	X =  100.000  mm,	Y =  199.000  mm,	Z =   15.000 mm,
	W =180.000 deg,	P =   0.000 deg,	R =    90.000 deg
};
P[9151]{
   GP1:
	UF : 1, UT : 1,		CONFIG : 'N U T, 0, 0, 1',
	X =  103.000  mm,	Y =  199.000  mm,	Z =   15.000 mm,
	W =180.000 deg,	P =   0.000 deg,	R =    90.000 deg
};
P[9152]{
   GP1:
	UF : 1, UT : 1,		CONFIG : 'N U T, 0, 0, 1',
	X =  103.000  mm,	Y =  199.000  mm,	Z =   0.600 mm,
	W =180.000 deg,	P =   0.000 deg,	R =    90.000 deg
};
P[9153]{
   GP1:
	UF : 1, UT : 1,		CONFIG : 'N U T, 0, 0, 1',
	X =  103.000  mm,	Y =  199.000  mm,	Z =   15.000 mm,
	W =180.000 deg,	P =   0.000 deg,	R =    90.000 deg
};
P[9154]{
   GP1:
	UF : 1, UT : 1,		CONFIG : 'N U T, 0, 0, 1',
	X =  106.000  mm,	Y =  199.000  mm,	Z =   15.000 mm,
	W =180.000 deg,	P =   0.000 deg,	R =    90.000 deg
};
P[9155]{
   GP1:
	UF : 1, UT : 1,		CONFIG : 'N U T, 0, 0, 1',
	X =  106.000  mm,	Y =  199.000  mm,	Z =   0.600 mm,
	W =180.000 deg,	P =   0.000 deg,	R =    90.000 deg
};
P[9156]{
   GP1:
	UF : 1, UT : 1,		CONFIG : 'N U T, 0, 0, 1',
	X =  106.000  mm,	Y =  199.000  mm,	Z =   15.000 mm,
	W =180.000 deg,	P =   0.000 deg,	R =    90.000 deg
};
P[9157]{
   GP1:
	UF : 1, UT : 1,		CONFIG : 'N U T, 0, 0, 1',
	X =  109.000  mm,	Y =  199.000  mm,	Z =   15.000 mm,
	W =180.000 deg,	P =   0.000 deg,	R =    90.000 deg
};
P[9158]{
   GP1:
	UF : 1, UT : 1,		CONFIG : 'N U T, 0, 0, 1',
	X =  109.000  mm,	Y =  199.000  mm,	Z =   0.600 mm,
	W =180.000 deg,	P =   0.000 deg,	R =    90.000 deg
};
P[9159]{
   GP1:
	UF : 1, UT : 1,		CONFIG : 'N U T, 0, 0, 1',
	X =  109.000  mm,	Y =  199.000  mm,	Z =   15.000 mm,
	W =180.000 deg,	P =   0.000 deg,	R =    90.000 deg
};
P[9160]{
   GP1:
	UF : 1, UT : 1,		CONFIG : 'N U T, 0, 0, 1',
	X =  112.000  mm,	Y =  199.000  mm,	Z =   15.000 mm,
	W =180.000 deg,	P =   0.000 deg,	R =    90.000 deg
};
P[9161]{
   GP1:
	UF : 1, UT : 1,		CONFIG : 'N U T, 0, 0, 1',
	X =  112.000  mm,	Y =  199.000  mm,	Z =   0.600 mm,
	W =180.000 deg,	P =   0.000 deg,	R =    90.000 deg
};
P[9162]{
   GP1:
	UF : 1, UT : 1,		CONFIG : 'N U T, 0, 0, 1',
	X =  112.000  mm,	Y =  199.000  mm,	Z =   15.000 mm,
	W =180.000 deg,	P =   0.000 deg,	R =    90.000 deg
};
P[9163]{
   GP1:
	UF : 1, UT : 1,		CONFIG : 'N U T, 0, 0, 1',
	X =  115.000  mm,	Y =  199.000  mm,	Z =   15.000 mm,
	W =180.000 deg,	P =   0.000 deg,	R =    90.000 deg
};
P[9164]{
   GP1:
	UF : 1, UT : 1,		CONFIG : 'N U T, 0, 0, 1',
	X =  115.000  mm,	Y =  199.000  mm,	Z =   0.600 mm,
	W =180.000 deg,	P =   0.000 deg,	R =    90.000 deg
};
P[9165]{
   GP1:
	UF : 1, UT : 1,		CONFIG : 'N U T, 0, 0, 1',
	X =  115.000  mm,	Y =  199.000  mm,	Z =   15.000 mm,
	W =180.000 deg,	P =   0.000 deg,	R =    90.000 deg
};
P[9166]{
   GP1:
	UF : 1, UT : 1,		CONFIG : 'N U T, 0, 0, 1',
	X =  118.000  mm,	Y =  199.000  mm,	Z =   15.000 mm,
	W =180.000 deg,	P =   0.000 deg,	R =    90.000 deg
};
P[9167]{
   GP1:
	UF : 1, UT : 1,		CONFIG : 'N U T, 0, 0, 1',
	X =  118.000  mm,	Y =  199.000  mm,	Z =   0.600 mm,
	W =180.000 deg,	P =   0.000 deg,	R =    90.000 deg
};
P[9168]{
   GP1:
	UF : 1, UT : 1,		CONFIG : 'N U T, 0, 0, 1',
	X =  118.000  mm,	Y =  199.000  mm,	Z =   15.000 mm,
	W =180.000 deg,	P =   0.000 deg,	R =    90.000 deg
};
P[9169]{
   GP1:
	UF : 1, UT : 1,		CONFIG : 'N U T, 0, 0, 1',
	X =  121.000  mm,	Y =  199.000  mm,	Z =   15.000 mm,
	W =180.000 deg,	P =   0.000 deg,	R =    90.000 deg
};
P[9170]{
   GP1:
	UF : 1, UT : 1,		CONFIG : 'N U T, 0, 0, 1',
	X =  121.000  mm,	Y =  199.000  mm,	Z =   0.600 mm,
	W =180.000 deg,	P =   0.000 deg,	R =    90.000 deg
};
P[9171]{
   GP1:
	UF : 1, UT : 1,		CONFIG : 'N U T, 0, 0, 1',
	X =  121.000  mm,	Y =  199.000  mm,	Z =   15.000 mm,
	W =180.000 deg,	P =   0.000 deg,	R =    90.000 deg
};
P[9172]{
   GP1:
	UF : 1, UT : 1,		CONFIG : 'N U T, 0, 0, 1',
	X =  124.000  mm,	Y =  199.000  mm,	Z =   15.000 mm,
	W =180.000 deg,	P =   0.000 deg,	R =    90.000 deg
};
P[9173]{
   GP1:
	UF : 1, UT : 1,		CONFIG : 'N U T, 0, 0, 1',
	X =  124.000  mm,	Y =  199.000  mm,	Z =   0.600 mm,
	W =180.000 deg,	P =   0.000 deg,	R =    90.000 deg
};
P[9174]{
   GP1:
	UF : 1, UT : 1,		CONFIG : 'N U T, 0, 0, 1',
	X =  124.000  mm,	Y =  199.000  mm,	Z =   15.000 mm,
	W =180.000 deg,	P =   0.000 deg,	R =    90.000 deg
};
P[9175]{
   GP1:
	UF : 1, UT : 1,		CONFIG : 'N U T, 0, 0, 1',
	X =  127.000  mm,	Y =  199.000  mm,	Z =   15.000 mm,
	W =180.000 deg,	P =   0.000 deg,	R =    90.000 deg
};
P[9176]{
   GP1:
	UF : 1, UT : 1,		CONFIG : 'N U T, 0, 0, 1',
	X =  127.000  mm,	Y =  199.000  mm,	Z =   0.600 mm,
	W =180.000 deg,	P =   0.000 deg,	R =    90.000 deg
};
P[9177]{
   GP1:
	UF : 1, UT : 1,		CONFIG : 'N U T, 0, 0, 1',
	X =  127.000  mm,	Y =  199.000  mm,	Z =   15.000 mm,
	W =180.000 deg,	P =   0.000 deg,	R =    90.000 deg
};
P[9178]{
   GP1:
	UF : 1, UT : 1,		CONFIG : 'N U T, 0, 0, 1',
	X =  130.000  mm,	Y =  199.000  mm,	Z =   15.000 mm,
	W =180.000 deg,	P =   0.000 deg,	R =    90.000 deg
};
P[9179]{
   GP1:
	UF : 1, UT : 1,		CONFIG : 'N U T, 0, 0, 1',
	X =  130.000  mm,	Y =  199.000  mm,	Z =   0.600 mm,
	W =180.000 deg,	P =   0.000 deg,	R =    90.000 deg
};
P[9180]{
   GP1:
	UF : 1, UT : 1,		CONFIG : 'N U T, 0, 0, 1',
	X =  130.000  mm,	Y =  199.000  mm,	Z =   15.000 mm,
	W =180.000 deg,	P =   0.000 deg,	R =    90.000 deg
};
P[9181]{
   GP1:
	UF : 1, UT : 1,		CONFIG : 'N U T, 0, 0, 1',
	X =  133.000  mm,	Y =  199.000  mm,	Z =   15.000 mm,
	W =180.000 deg,	P =   0.000 deg,	R =    90.000 deg
};
P[9182]{
   GP1:
	UF : 1, UT : 1,		CONFIG : 'N U T, 0, 0, 1',
	X =  133.000  mm,	Y =  199.000  mm,	Z =   0.600 mm,
	W =180.000 deg,	P =   0.000 deg,	R =    90.000 deg
};
P[9183]{
   GP1:
	UF : 1, UT : 1,		CONFIG : 'N U T, 0, 0, 1',
	X =  133.000  mm,	Y =  199.000  mm,	Z =   15.000 mm,
	W =180.000 deg,	P =   0.000 deg,	R =    90.000 deg
};
P[9184]{
   GP1:
	UF : 1, UT : 1,		CONFIG : 'N U T, 0, 0, 1',
	X =  136.000  mm,	Y =  199.000  mm,	Z =   15.000 mm,
	W =180.000 deg,	P =   0.000 deg,	R =    90.000 deg
};
P[9185]{
   GP1:
	UF : 1, UT : 1,		CONFIG : 'N U T, 0, 0, 1',
	X =  136.000  mm,	Y =  199.000  mm,	Z =   0.600 mm,
	W =180.000 deg,	P =   0.000 deg,	R =    90.000 deg
};
P[9186]{
   GP1:
	UF : 1, UT : 1,		CONFIG : 'N U T, 0, 0, 1',
	X =  136.000  mm,	Y =  199.000  mm,	Z =   15.000 mm,
	W =180.000 deg,	P =   0.000 deg,	R =    90.000 deg
};
P[9187]{
   GP1:
	UF : 1, UT : 1,		CONFIG : 'N U T, 0, 0, 1',
	X =  139.000  mm,	Y =  199.000  mm,	Z =   15.000 mm,
	W =180.000 deg,	P =   0.000 deg,	R =    90.000 deg
};
P[9188]{
   GP1:
	UF : 1, UT : 1,		CONFIG : 'N U T, 0, 0, 1',
	X =  139.000  mm,	Y =  199.000  mm,	Z =   0.600 mm,
	W =180.000 deg,	P =   0.000 deg,	R =    90.000 deg
};
P[9189]{
   GP1:
	UF : 1, UT : 1,		CONFIG : 'N U T, 0, 0, 1',
	X =  139.000  mm,	Y =  199.000  mm,	Z =   15.000 mm,
	W =180.000 deg,	P =   0.000 deg,	R =    90.000 deg
};
P[9190]{
   GP1:
	UF : 1, UT : 1,		CONFIG : 'N U T, 0, 0, 1',
	X =  142.000  mm,	Y =  199.000  mm,	Z =   15.000 mm,
	W =180.000 deg,	P =   0.000 deg,	R =    90.000 deg
};
P[9191]{
   GP1:
	UF : 1, UT : 1,		CONFIG : 'N U T, 0, 0, 1',
	X =  142.000  mm,	Y =  199.000  mm,	Z =   0.600 mm,
	W =180.000 deg,	P =   0.000 deg,	R =    90.000 deg
};
P[9192]{
   GP1:
	UF : 1, UT : 1,		CONFIG : 'N U T, 0, 0, 1',
	X =  142.000  mm,	Y =  199.000  mm,	Z =   15.000 mm,
	W =180.000 deg,	P =   0.000 deg,	R =    90.000 deg
};
P[9193]{
   GP1:
	UF : 1, UT : 1,		CONFIG : 'N U T, 0, 0, 1',
	X =  145.000  mm,	Y =  199.000  mm,	Z =   15.000 mm,
	W =180.000 deg,	P =   0.000 deg,	R =    90.000 deg
};
P[9194]{
   GP1:
	UF : 1, UT : 1,		CONFIG : 'N U T, 0, 0, 1',
	X =  145.000  mm,	Y =  199.000  mm,	Z =   0.600 mm,
	W =180.000 deg,	P =   0.000 deg,	R =    90.000 deg
};
P[9195]{
   GP1:
	UF : 1, UT : 1,		CONFIG : 'N U T, 0, 0, 1',
	X =  145.000  mm,	Y =  199.000  mm,	Z =   15.000 mm,
	W =180.000 deg,	P =   0.000 deg,	R =    90.000 deg
};
P[9196]{
   GP1:
	UF : 1, UT : 1,		CONFIG : 'N U T, 0, 0, 1',
	X =  148.000  mm,	Y =  199.000  mm,	Z =   15.000 mm,
	W =180.000 deg,	P =   0.000 deg,	R =    90.000 deg
};
P[9197]{
   GP1:
	UF : 1, UT : 1,		CONFIG : 'N U T, 0, 0, 1',
	X =  148.000  mm,	Y =  199.000  mm,	Z =   0.600 mm,
	W =180.000 deg,	P =   0.000 deg,	R =    90.000 deg
};
P[9198]{
   GP1:
	UF : 1, UT : 1,		CONFIG : 'N U T, 0, 0, 1',
	X =  148.000  mm,	Y =  199.000  mm,	Z =   15.000 mm,
	W =180.000 deg,	P =   0.000 deg,	R =    90.000 deg
};
P[9199]{
   GP1:
	UF : 1, UT : 1,		CONFIG : 'N U T, 0, 0, 1',
	X =  151.000  mm,	Y =  199.000  mm,	Z =   15.000 mm,
	W =180.000 deg,	P =   0.000 deg,	R =    90.000 deg
};
P[9200]{
   GP1:
	UF : 1, UT : 1,		CONFIG : 'N U T, 0, 0, 1',
	X =  151.000  mm,	Y =  199.000  mm,	Z =   0.600 mm,
	W =180.000 deg,	P =   0.000 deg,	R =    90.000 deg
};
P[9201]{
   GP1:
	UF : 1, UT : 1,		CONFIG : 'N U T, 0, 0, 1',
	X =  151.000  mm,	Y =  199.000  mm,	Z =   15.000 mm,
	W =180.000 deg,	P =   0.000 deg,	R =    90.000 deg
};
P[9202]{
   GP1:
	UF : 1, UT : 1,		CONFIG : 'N U T, 0, 0, 1',
	X =  154.000  mm,	Y =  199.000  mm,	Z =   15.000 mm,
	W =180.000 deg,	P =   0.000 deg,	R =    90.000 deg
};
P[9203]{
   GP1:
	UF : 1, UT : 1,		CONFIG : 'N U T, 0, 0, 1',
	X =  154.000  mm,	Y =  199.000  mm,	Z =   0.600 mm,
	W =180.000 deg,	P =   0.000 deg,	R =    90.000 deg
};
P[9204]{
   GP1:
	UF : 1, UT : 1,		CONFIG : 'N U T, 0, 0, 1',
	X =  154.000  mm,	Y =  199.000  mm,	Z =   15.000 mm,
	W =180.000 deg,	P =   0.000 deg,	R =    90.000 deg
};
P[9205]{
   GP1:
	UF : 1, UT : 1,		CONFIG : 'N U T, 0, 0, 1',
	X =  157.000  mm,	Y =  199.000  mm,	Z =   15.000 mm,
	W =180.000 deg,	P =   0.000 deg,	R =    90.000 deg
};
P[9206]{
   GP1:
	UF : 1, UT : 1,		CONFIG : 'N U T, 0, 0, 1',
	X =  157.000  mm,	Y =  199.000  mm,	Z =   0.600 mm,
	W =180.000 deg,	P =   0.000 deg,	R =    90.000 deg
};
P[9207]{
   GP1:
	UF : 1, UT : 1,		CONFIG : 'N U T, 0, 0, 1',
	X =  157.000  mm,	Y =  199.000  mm,	Z =   15.000 mm,
	W =180.000 deg,	P =   0.000 deg,	R =    90.000 deg
};
P[9208]{
   GP1:
	UF : 1, UT : 1,		CONFIG : 'N U T, 0, 0, 1',
	X =  160.000  mm,	Y =  199.000  mm,	Z =   15.000 mm,
	W =180.000 deg,	P =   0.000 deg,	R =    90.000 deg
};
P[9209]{
   GP1:
	UF : 1, UT : 1,		CONFIG : 'N U T, 0, 0, 1',
	X =  160.000  mm,	Y =  199.000  mm,	Z =   0.600 mm,
	W =180.000 deg,	P =   0.000 deg,	R =    90.000 deg
};
P[9210]{
   GP1:
	UF : 1, UT : 1,		CONFIG : 'N U T, 0, 0, 1',
	X =  160.000  mm,	Y =  199.000  mm,	Z =   15.000 mm,
	W =180.000 deg,	P =   0.000 deg,	R =    90.000 deg
};
P[9211]{
   GP1:
	UF : 1, UT : 1,		CONFIG : 'N U T, 0, 0, 1',
	X =  163.000  mm,	Y =  199.000  mm,	Z =   15.000 mm,
	W =180.000 deg,	P =   0.000 deg,	R =    90.000 deg
};
P[9212]{
   GP1:
	UF : 1, UT : 1,		CONFIG : 'N U T, 0, 0, 1',
	X =  163.000  mm,	Y =  199.000  mm,	Z =   0.600 mm,
	W =180.000 deg,	P =   0.000 deg,	R =    90.000 deg
};
P[9213]{
   GP1:
	UF : 1, UT : 1,		CONFIG : 'N U T, 0, 0, 1',
	X =  163.000  mm,	Y =  199.000  mm,	Z =   15.000 mm,
	W =180.000 deg,	P =   0.000 deg,	R =    90.000 deg
};
P[9214]{
   GP1:
	UF : 1, UT : 1,		CONFIG : 'N U T, 0, 0, 1',
	X =  166.000  mm,	Y =  199.000  mm,	Z =   15.000 mm,
	W =180.000 deg,	P =   0.000 deg,	R =    90.000 deg
};
P[9215]{
   GP1:
	UF : 1, UT : 1,		CONFIG : 'N U T, 0, 0, 1',
	X =  166.000  mm,	Y =  199.000  mm,	Z =   0.600 mm,
	W =180.000 deg,	P =   0.000 deg,	R =    90.000 deg
};
P[9216]{
   GP1:
	UF : 1, UT : 1,		CONFIG : 'N U T, 0, 0, 1',
	X =  166.000  mm,	Y =  199.000  mm,	Z =   15.000 mm,
	W =180.000 deg,	P =   0.000 deg,	R =    90.000 deg
};
P[9217]{
   GP1:
	UF : 1, UT : 1,		CONFIG : 'N U T, 0, 0, 1',
	X =  169.000  mm,	Y =  199.000  mm,	Z =   15.000 mm,
	W =180.000 deg,	P =   0.000 deg,	R =    90.000 deg
};
P[9218]{
   GP1:
	UF : 1, UT : 1,		CONFIG : 'N U T, 0, 0, 1',
	X =  169.000  mm,	Y =  199.000  mm,	Z =   0.600 mm,
	W =180.000 deg,	P =   0.000 deg,	R =    90.000 deg
};
P[9219]{
   GP1:
	UF : 1, UT : 1,		CONFIG : 'N U T, 0, 0, 1',
	X =  169.000  mm,	Y =  199.000  mm,	Z =   15.000 mm,
	W =180.000 deg,	P =   0.000 deg,	R =    90.000 deg
};
P[9220]{
   GP1:
	UF : 1, UT : 1,		CONFIG : 'N U T, 0, 0, 1',
	X =  172.000  mm,	Y =  199.000  mm,	Z =   15.000 mm,
	W =180.000 deg,	P =   0.000 deg,	R =    90.000 deg
};
P[9221]{
   GP1:
	UF : 1, UT : 1,		CONFIG : 'N U T, 0, 0, 1',
	X =  172.000  mm,	Y =  199.000  mm,	Z =   0.600 mm,
	W =180.000 deg,	P =   0.000 deg,	R =    90.000 deg
};
P[9222]{
   GP1:
	UF : 1, UT : 1,		CONFIG : 'N U T, 0, 0, 1',
	X =  172.000  mm,	Y =  199.000  mm,	Z =   15.000 mm,
	W =180.000 deg,	P =   0.000 deg,	R =    90.000 deg
};
P[9223]{
   GP1:
	UF : 1, UT : 1,		CONFIG : 'N U T, 0, 0, 1',
	X =  175.000  mm,	Y =  199.000  mm,	Z =   15.000 mm,
	W =180.000 deg,	P =   0.000 deg,	R =    90.000 deg
};
P[9224]{
   GP1:
	UF : 1, UT : 1,		CONFIG : 'N U T, 0, 0, 1',
	X =  175.000  mm,	Y =  199.000  mm,	Z =   0.600 mm,
	W =180.000 deg,	P =   0.000 deg,	R =    90.000 deg
};
P[9225]{
   GP1:
	UF : 1, UT : 1,		CONFIG : 'N U T, 0, 0, 1',
	X =  175.000  mm,	Y =  199.000  mm,	Z =   15.000 mm,
	W =180.000 deg,	P =   0.000 deg,	R =    90.000 deg
};
P[9226]{
   GP1:
	UF : 1, UT : 1,		CONFIG : 'N U T, 0, 0, 1',
	X =  178.000  mm,	Y =  199.000  mm,	Z =   15.000 mm,
	W =180.000 deg,	P =   0.000 deg,	R =    90.000 deg
};
P[9227]{
   GP1:
	UF : 1, UT : 1,		CONFIG : 'N U T, 0, 0, 1',
	X =  178.000  mm,	Y =  199.000  mm,	Z =   0.600 mm,
	W =180.000 deg,	P =   0.000 deg,	R =    90.000 deg
};
P[9228]{
   GP1:
	UF : 1, UT : 1,		CONFIG : 'N U T, 0, 0, 1',
	X =  178.000  mm,	Y =  199.000  mm,	Z =   15.000 mm,
	W =180.000 deg,	P =   0.000 deg,	R =    90.000 deg
};
P[9229]{
   GP1:
	UF : 1, UT : 1,		CONFIG : 'N U T, 0, 0, 1',
	X =  1.000  mm,	Y =  202.000  mm,	Z =   15.000 mm,
	W =180.000 deg,	P =   0.000 deg,	R =    90.000 deg
};
P[9230]{
   GP1:
	UF : 1, UT : 1,		CONFIG : 'N U T, 0, 0, 1',
	X =  1.000  mm,	Y =  202.000  mm,	Z =   0.600 mm,
	W =180.000 deg,	P =   0.000 deg,	R =    90.000 deg
};
P[9231]{
   GP1:
	UF : 1, UT : 1,		CONFIG : 'N U T, 0, 0, 1',
	X =  1.000  mm,	Y =  202.000  mm,	Z =   15.000 mm,
	W =180.000 deg,	P =   0.000 deg,	R =    90.000 deg
};
P[9232]{
   GP1:
	UF : 1, UT : 1,		CONFIG : 'N U T, 0, 0, 1',
	X =  4.000  mm,	Y =  202.000  mm,	Z =   15.000 mm,
	W =180.000 deg,	P =   0.000 deg,	R =    90.000 deg
};
P[9233]{
   GP1:
	UF : 1, UT : 1,		CONFIG : 'N U T, 0, 0, 1',
	X =  4.000  mm,	Y =  202.000  mm,	Z =   0.600 mm,
	W =180.000 deg,	P =   0.000 deg,	R =    90.000 deg
};
P[9234]{
   GP1:
	UF : 1, UT : 1,		CONFIG : 'N U T, 0, 0, 1',
	X =  4.000  mm,	Y =  202.000  mm,	Z =   15.000 mm,
	W =180.000 deg,	P =   0.000 deg,	R =    90.000 deg
};
P[9235]{
   GP1:
	UF : 1, UT : 1,		CONFIG : 'N U T, 0, 0, 1',
	X =  7.000  mm,	Y =  202.000  mm,	Z =   15.000 mm,
	W =180.000 deg,	P =   0.000 deg,	R =    90.000 deg
};
P[9236]{
   GP1:
	UF : 1, UT : 1,		CONFIG : 'N U T, 0, 0, 1',
	X =  7.000  mm,	Y =  202.000  mm,	Z =   0.600 mm,
	W =180.000 deg,	P =   0.000 deg,	R =    90.000 deg
};
P[9237]{
   GP1:
	UF : 1, UT : 1,		CONFIG : 'N U T, 0, 0, 1',
	X =  7.000  mm,	Y =  202.000  mm,	Z =   15.000 mm,
	W =180.000 deg,	P =   0.000 deg,	R =    90.000 deg
};
P[9238]{
   GP1:
	UF : 1, UT : 1,		CONFIG : 'N U T, 0, 0, 1',
	X =  10.000  mm,	Y =  202.000  mm,	Z =   15.000 mm,
	W =180.000 deg,	P =   0.000 deg,	R =    90.000 deg
};
P[9239]{
   GP1:
	UF : 1, UT : 1,		CONFIG : 'N U T, 0, 0, 1',
	X =  10.000  mm,	Y =  202.000  mm,	Z =   0.600 mm,
	W =180.000 deg,	P =   0.000 deg,	R =    90.000 deg
};
P[9240]{
   GP1:
	UF : 1, UT : 1,		CONFIG : 'N U T, 0, 0, 1',
	X =  10.000  mm,	Y =  202.000  mm,	Z =   15.000 mm,
	W =180.000 deg,	P =   0.000 deg,	R =    90.000 deg
};
P[9241]{
   GP1:
	UF : 1, UT : 1,		CONFIG : 'N U T, 0, 0, 1',
	X =  13.000  mm,	Y =  202.000  mm,	Z =   15.000 mm,
	W =180.000 deg,	P =   0.000 deg,	R =    90.000 deg
};
P[9242]{
   GP1:
	UF : 1, UT : 1,		CONFIG : 'N U T, 0, 0, 1',
	X =  13.000  mm,	Y =  202.000  mm,	Z =   0.600 mm,
	W =180.000 deg,	P =   0.000 deg,	R =    90.000 deg
};
P[9243]{
   GP1:
	UF : 1, UT : 1,		CONFIG : 'N U T, 0, 0, 1',
	X =  13.000  mm,	Y =  202.000  mm,	Z =   15.000 mm,
	W =180.000 deg,	P =   0.000 deg,	R =    90.000 deg
};
P[9244]{
   GP1:
	UF : 1, UT : 1,		CONFIG : 'N U T, 0, 0, 1',
	X =  16.000  mm,	Y =  202.000  mm,	Z =   15.000 mm,
	W =180.000 deg,	P =   0.000 deg,	R =    90.000 deg
};
P[9245]{
   GP1:
	UF : 1, UT : 1,		CONFIG : 'N U T, 0, 0, 1',
	X =  16.000  mm,	Y =  202.000  mm,	Z =   0.600 mm,
	W =180.000 deg,	P =   0.000 deg,	R =    90.000 deg
};
P[9246]{
   GP1:
	UF : 1, UT : 1,		CONFIG : 'N U T, 0, 0, 1',
	X =  16.000  mm,	Y =  202.000  mm,	Z =   15.000 mm,
	W =180.000 deg,	P =   0.000 deg,	R =    90.000 deg
};
P[9247]{
   GP1:
	UF : 1, UT : 1,		CONFIG : 'N U T, 0, 0, 1',
	X =  19.000  mm,	Y =  202.000  mm,	Z =   15.000 mm,
	W =180.000 deg,	P =   0.000 deg,	R =    90.000 deg
};
P[9248]{
   GP1:
	UF : 1, UT : 1,		CONFIG : 'N U T, 0, 0, 1',
	X =  19.000  mm,	Y =  202.000  mm,	Z =   0.600 mm,
	W =180.000 deg,	P =   0.000 deg,	R =    90.000 deg
};
P[9249]{
   GP1:
	UF : 1, UT : 1,		CONFIG : 'N U T, 0, 0, 1',
	X =  19.000  mm,	Y =  202.000  mm,	Z =   15.000 mm,
	W =180.000 deg,	P =   0.000 deg,	R =    90.000 deg
};
P[9250]{
   GP1:
	UF : 1, UT : 1,		CONFIG : 'N U T, 0, 0, 1',
	X =  22.000  mm,	Y =  202.000  mm,	Z =   15.000 mm,
	W =180.000 deg,	P =   0.000 deg,	R =    90.000 deg
};
P[9251]{
   GP1:
	UF : 1, UT : 1,		CONFIG : 'N U T, 0, 0, 1',
	X =  22.000  mm,	Y =  202.000  mm,	Z =   0.600 mm,
	W =180.000 deg,	P =   0.000 deg,	R =    90.000 deg
};
P[9252]{
   GP1:
	UF : 1, UT : 1,		CONFIG : 'N U T, 0, 0, 1',
	X =  22.000  mm,	Y =  202.000  mm,	Z =   15.000 mm,
	W =180.000 deg,	P =   0.000 deg,	R =    90.000 deg
};
P[9253]{
   GP1:
	UF : 1, UT : 1,		CONFIG : 'N U T, 0, 0, 1',
	X =  25.000  mm,	Y =  202.000  mm,	Z =   15.000 mm,
	W =180.000 deg,	P =   0.000 deg,	R =    90.000 deg
};
P[9254]{
   GP1:
	UF : 1, UT : 1,		CONFIG : 'N U T, 0, 0, 1',
	X =  25.000  mm,	Y =  202.000  mm,	Z =   0.600 mm,
	W =180.000 deg,	P =   0.000 deg,	R =    90.000 deg
};
P[9255]{
   GP1:
	UF : 1, UT : 1,		CONFIG : 'N U T, 0, 0, 1',
	X =  25.000  mm,	Y =  202.000  mm,	Z =   15.000 mm,
	W =180.000 deg,	P =   0.000 deg,	R =    90.000 deg
};
P[9256]{
   GP1:
	UF : 1, UT : 1,		CONFIG : 'N U T, 0, 0, 1',
	X =  28.000  mm,	Y =  202.000  mm,	Z =   15.000 mm,
	W =180.000 deg,	P =   0.000 deg,	R =    90.000 deg
};
P[9257]{
   GP1:
	UF : 1, UT : 1,		CONFIG : 'N U T, 0, 0, 1',
	X =  28.000  mm,	Y =  202.000  mm,	Z =   0.600 mm,
	W =180.000 deg,	P =   0.000 deg,	R =    90.000 deg
};
P[9258]{
   GP1:
	UF : 1, UT : 1,		CONFIG : 'N U T, 0, 0, 1',
	X =  28.000  mm,	Y =  202.000  mm,	Z =   15.000 mm,
	W =180.000 deg,	P =   0.000 deg,	R =    90.000 deg
};
P[9259]{
   GP1:
	UF : 1, UT : 1,		CONFIG : 'N U T, 0, 0, 1',
	X =  31.000  mm,	Y =  202.000  mm,	Z =   15.000 mm,
	W =180.000 deg,	P =   0.000 deg,	R =    90.000 deg
};
P[9260]{
   GP1:
	UF : 1, UT : 1,		CONFIG : 'N U T, 0, 0, 1',
	X =  31.000  mm,	Y =  202.000  mm,	Z =   0.600 mm,
	W =180.000 deg,	P =   0.000 deg,	R =    90.000 deg
};
P[9261]{
   GP1:
	UF : 1, UT : 1,		CONFIG : 'N U T, 0, 0, 1',
	X =  31.000  mm,	Y =  202.000  mm,	Z =   15.000 mm,
	W =180.000 deg,	P =   0.000 deg,	R =    90.000 deg
};
P[9262]{
   GP1:
	UF : 1, UT : 1,		CONFIG : 'N U T, 0, 0, 1',
	X =  34.000  mm,	Y =  202.000  mm,	Z =   15.000 mm,
	W =180.000 deg,	P =   0.000 deg,	R =    90.000 deg
};
P[9263]{
   GP1:
	UF : 1, UT : 1,		CONFIG : 'N U T, 0, 0, 1',
	X =  34.000  mm,	Y =  202.000  mm,	Z =   0.600 mm,
	W =180.000 deg,	P =   0.000 deg,	R =    90.000 deg
};
P[9264]{
   GP1:
	UF : 1, UT : 1,		CONFIG : 'N U T, 0, 0, 1',
	X =  34.000  mm,	Y =  202.000  mm,	Z =   15.000 mm,
	W =180.000 deg,	P =   0.000 deg,	R =    90.000 deg
};
P[9265]{
   GP1:
	UF : 1, UT : 1,		CONFIG : 'N U T, 0, 0, 1',
	X =  37.000  mm,	Y =  202.000  mm,	Z =   15.000 mm,
	W =180.000 deg,	P =   0.000 deg,	R =    90.000 deg
};
P[9266]{
   GP1:
	UF : 1, UT : 1,		CONFIG : 'N U T, 0, 0, 1',
	X =  37.000  mm,	Y =  202.000  mm,	Z =   0.600 mm,
	W =180.000 deg,	P =   0.000 deg,	R =    90.000 deg
};
P[9267]{
   GP1:
	UF : 1, UT : 1,		CONFIG : 'N U T, 0, 0, 1',
	X =  37.000  mm,	Y =  202.000  mm,	Z =   15.000 mm,
	W =180.000 deg,	P =   0.000 deg,	R =    90.000 deg
};
P[9268]{
   GP1:
	UF : 1, UT : 1,		CONFIG : 'N U T, 0, 0, 1',
	X =  40.000  mm,	Y =  202.000  mm,	Z =   15.000 mm,
	W =180.000 deg,	P =   0.000 deg,	R =    90.000 deg
};
P[9269]{
   GP1:
	UF : 1, UT : 1,		CONFIG : 'N U T, 0, 0, 1',
	X =  40.000  mm,	Y =  202.000  mm,	Z =   0.600 mm,
	W =180.000 deg,	P =   0.000 deg,	R =    90.000 deg
};
P[9270]{
   GP1:
	UF : 1, UT : 1,		CONFIG : 'N U T, 0, 0, 1',
	X =  40.000  mm,	Y =  202.000  mm,	Z =   15.000 mm,
	W =180.000 deg,	P =   0.000 deg,	R =    90.000 deg
};
P[9271]{
   GP1:
	UF : 1, UT : 1,		CONFIG : 'N U T, 0, 0, 1',
	X =  43.000  mm,	Y =  202.000  mm,	Z =   15.000 mm,
	W =180.000 deg,	P =   0.000 deg,	R =    90.000 deg
};
P[9272]{
   GP1:
	UF : 1, UT : 1,		CONFIG : 'N U T, 0, 0, 1',
	X =  43.000  mm,	Y =  202.000  mm,	Z =   0.600 mm,
	W =180.000 deg,	P =   0.000 deg,	R =    90.000 deg
};
P[9273]{
   GP1:
	UF : 1, UT : 1,		CONFIG : 'N U T, 0, 0, 1',
	X =  43.000  mm,	Y =  202.000  mm,	Z =   15.000 mm,
	W =180.000 deg,	P =   0.000 deg,	R =    90.000 deg
};
P[9274]{
   GP1:
	UF : 1, UT : 1,		CONFIG : 'N U T, 0, 0, 1',
	X =  46.000  mm,	Y =  202.000  mm,	Z =   15.000 mm,
	W =180.000 deg,	P =   0.000 deg,	R =    90.000 deg
};
P[9275]{
   GP1:
	UF : 1, UT : 1,		CONFIG : 'N U T, 0, 0, 1',
	X =  46.000  mm,	Y =  202.000  mm,	Z =   0.600 mm,
	W =180.000 deg,	P =   0.000 deg,	R =    90.000 deg
};
P[9276]{
   GP1:
	UF : 1, UT : 1,		CONFIG : 'N U T, 0, 0, 1',
	X =  46.000  mm,	Y =  202.000  mm,	Z =   15.000 mm,
	W =180.000 deg,	P =   0.000 deg,	R =    90.000 deg
};
P[9277]{
   GP1:
	UF : 1, UT : 1,		CONFIG : 'N U T, 0, 0, 1',
	X =  49.000  mm,	Y =  202.000  mm,	Z =   15.000 mm,
	W =180.000 deg,	P =   0.000 deg,	R =    90.000 deg
};
P[9278]{
   GP1:
	UF : 1, UT : 1,		CONFIG : 'N U T, 0, 0, 1',
	X =  49.000  mm,	Y =  202.000  mm,	Z =   0.600 mm,
	W =180.000 deg,	P =   0.000 deg,	R =    90.000 deg
};
P[9279]{
   GP1:
	UF : 1, UT : 1,		CONFIG : 'N U T, 0, 0, 1',
	X =  49.000  mm,	Y =  202.000  mm,	Z =   15.000 mm,
	W =180.000 deg,	P =   0.000 deg,	R =    90.000 deg
};
P[9280]{
   GP1:
	UF : 1, UT : 1,		CONFIG : 'N U T, 0, 0, 1',
	X =  52.000  mm,	Y =  202.000  mm,	Z =   15.000 mm,
	W =180.000 deg,	P =   0.000 deg,	R =    90.000 deg
};
P[9281]{
   GP1:
	UF : 1, UT : 1,		CONFIG : 'N U T, 0, 0, 1',
	X =  52.000  mm,	Y =  202.000  mm,	Z =   0.600 mm,
	W =180.000 deg,	P =   0.000 deg,	R =    90.000 deg
};
P[9282]{
   GP1:
	UF : 1, UT : 1,		CONFIG : 'N U T, 0, 0, 1',
	X =  52.000  mm,	Y =  202.000  mm,	Z =   15.000 mm,
	W =180.000 deg,	P =   0.000 deg,	R =    90.000 deg
};
P[9283]{
   GP1:
	UF : 1, UT : 1,		CONFIG : 'N U T, 0, 0, 1',
	X =  55.000  mm,	Y =  202.000  mm,	Z =   15.000 mm,
	W =180.000 deg,	P =   0.000 deg,	R =    90.000 deg
};
P[9284]{
   GP1:
	UF : 1, UT : 1,		CONFIG : 'N U T, 0, 0, 1',
	X =  55.000  mm,	Y =  202.000  mm,	Z =   0.600 mm,
	W =180.000 deg,	P =   0.000 deg,	R =    90.000 deg
};
P[9285]{
   GP1:
	UF : 1, UT : 1,		CONFIG : 'N U T, 0, 0, 1',
	X =  55.000  mm,	Y =  202.000  mm,	Z =   15.000 mm,
	W =180.000 deg,	P =   0.000 deg,	R =    90.000 deg
};
P[9286]{
   GP1:
	UF : 1, UT : 1,		CONFIG : 'N U T, 0, 0, 1',
	X =  58.000  mm,	Y =  202.000  mm,	Z =   15.000 mm,
	W =180.000 deg,	P =   0.000 deg,	R =    90.000 deg
};
P[9287]{
   GP1:
	UF : 1, UT : 1,		CONFIG : 'N U T, 0, 0, 1',
	X =  58.000  mm,	Y =  202.000  mm,	Z =   0.600 mm,
	W =180.000 deg,	P =   0.000 deg,	R =    90.000 deg
};
P[9288]{
   GP1:
	UF : 1, UT : 1,		CONFIG : 'N U T, 0, 0, 1',
	X =  58.000  mm,	Y =  202.000  mm,	Z =   15.000 mm,
	W =180.000 deg,	P =   0.000 deg,	R =    90.000 deg
};
P[9289]{
   GP1:
	UF : 1, UT : 1,		CONFIG : 'N U T, 0, 0, 1',
	X =  61.000  mm,	Y =  202.000  mm,	Z =   15.000 mm,
	W =180.000 deg,	P =   0.000 deg,	R =    90.000 deg
};
P[9290]{
   GP1:
	UF : 1, UT : 1,		CONFIG : 'N U T, 0, 0, 1',
	X =  61.000  mm,	Y =  202.000  mm,	Z =   0.600 mm,
	W =180.000 deg,	P =   0.000 deg,	R =    90.000 deg
};
P[9291]{
   GP1:
	UF : 1, UT : 1,		CONFIG : 'N U T, 0, 0, 1',
	X =  61.000  mm,	Y =  202.000  mm,	Z =   15.000 mm,
	W =180.000 deg,	P =   0.000 deg,	R =    90.000 deg
};
P[9292]{
   GP1:
	UF : 1, UT : 1,		CONFIG : 'N U T, 0, 0, 1',
	X =  64.000  mm,	Y =  202.000  mm,	Z =   15.000 mm,
	W =180.000 deg,	P =   0.000 deg,	R =    90.000 deg
};
P[9293]{
   GP1:
	UF : 1, UT : 1,		CONFIG : 'N U T, 0, 0, 1',
	X =  64.000  mm,	Y =  202.000  mm,	Z =   0.600 mm,
	W =180.000 deg,	P =   0.000 deg,	R =    90.000 deg
};
P[9294]{
   GP1:
	UF : 1, UT : 1,		CONFIG : 'N U T, 0, 0, 1',
	X =  64.000  mm,	Y =  202.000  mm,	Z =   15.000 mm,
	W =180.000 deg,	P =   0.000 deg,	R =    90.000 deg
};
P[9295]{
   GP1:
	UF : 1, UT : 1,		CONFIG : 'N U T, 0, 0, 1',
	X =  67.000  mm,	Y =  202.000  mm,	Z =   15.000 mm,
	W =180.000 deg,	P =   0.000 deg,	R =    90.000 deg
};
P[9296]{
   GP1:
	UF : 1, UT : 1,		CONFIG : 'N U T, 0, 0, 1',
	X =  67.000  mm,	Y =  202.000  mm,	Z =   0.600 mm,
	W =180.000 deg,	P =   0.000 deg,	R =    90.000 deg
};
P[9297]{
   GP1:
	UF : 1, UT : 1,		CONFIG : 'N U T, 0, 0, 1',
	X =  67.000  mm,	Y =  202.000  mm,	Z =   15.000 mm,
	W =180.000 deg,	P =   0.000 deg,	R =    90.000 deg
};
P[9298]{
   GP1:
	UF : 1, UT : 1,		CONFIG : 'N U T, 0, 0, 1',
	X =  70.000  mm,	Y =  202.000  mm,	Z =   15.000 mm,
	W =180.000 deg,	P =   0.000 deg,	R =    90.000 deg
};
P[9299]{
   GP1:
	UF : 1, UT : 1,		CONFIG : 'N U T, 0, 0, 1',
	X =  70.000  mm,	Y =  202.000  mm,	Z =   0.600 mm,
	W =180.000 deg,	P =   0.000 deg,	R =    90.000 deg
};
P[9300]{
   GP1:
	UF : 1, UT : 1,		CONFIG : 'N U T, 0, 0, 1',
	X =  70.000  mm,	Y =  202.000  mm,	Z =   15.000 mm,
	W =180.000 deg,	P =   0.000 deg,	R =    90.000 deg
};
P[9301]{
   GP1:
	UF : 1, UT : 1,		CONFIG : 'N U T, 0, 0, 1',
	X =  73.000  mm,	Y =  202.000  mm,	Z =   15.000 mm,
	W =180.000 deg,	P =   0.000 deg,	R =    90.000 deg
};
P[9302]{
   GP1:
	UF : 1, UT : 1,		CONFIG : 'N U T, 0, 0, 1',
	X =  73.000  mm,	Y =  202.000  mm,	Z =   0.600 mm,
	W =180.000 deg,	P =   0.000 deg,	R =    90.000 deg
};
P[9303]{
   GP1:
	UF : 1, UT : 1,		CONFIG : 'N U T, 0, 0, 1',
	X =  73.000  mm,	Y =  202.000  mm,	Z =   15.000 mm,
	W =180.000 deg,	P =   0.000 deg,	R =    90.000 deg
};
P[9304]{
   GP1:
	UF : 1, UT : 1,		CONFIG : 'N U T, 0, 0, 1',
	X =  76.000  mm,	Y =  202.000  mm,	Z =   15.000 mm,
	W =180.000 deg,	P =   0.000 deg,	R =    90.000 deg
};
P[9305]{
   GP1:
	UF : 1, UT : 1,		CONFIG : 'N U T, 0, 0, 1',
	X =  76.000  mm,	Y =  202.000  mm,	Z =   0.600 mm,
	W =180.000 deg,	P =   0.000 deg,	R =    90.000 deg
};
P[9306]{
   GP1:
	UF : 1, UT : 1,		CONFIG : 'N U T, 0, 0, 1',
	X =  76.000  mm,	Y =  202.000  mm,	Z =   15.000 mm,
	W =180.000 deg,	P =   0.000 deg,	R =    90.000 deg
};
P[9307]{
   GP1:
	UF : 1, UT : 1,		CONFIG : 'N U T, 0, 0, 1',
	X =  79.000  mm,	Y =  202.000  mm,	Z =   15.000 mm,
	W =180.000 deg,	P =   0.000 deg,	R =    90.000 deg
};
P[9308]{
   GP1:
	UF : 1, UT : 1,		CONFIG : 'N U T, 0, 0, 1',
	X =  79.000  mm,	Y =  202.000  mm,	Z =   0.600 mm,
	W =180.000 deg,	P =   0.000 deg,	R =    90.000 deg
};
P[9309]{
   GP1:
	UF : 1, UT : 1,		CONFIG : 'N U T, 0, 0, 1',
	X =  79.000  mm,	Y =  202.000  mm,	Z =   15.000 mm,
	W =180.000 deg,	P =   0.000 deg,	R =    90.000 deg
};
P[9310]{
   GP1:
	UF : 1, UT : 1,		CONFIG : 'N U T, 0, 0, 1',
	X =  82.000  mm,	Y =  202.000  mm,	Z =   15.000 mm,
	W =180.000 deg,	P =   0.000 deg,	R =    90.000 deg
};
P[9311]{
   GP1:
	UF : 1, UT : 1,		CONFIG : 'N U T, 0, 0, 1',
	X =  82.000  mm,	Y =  202.000  mm,	Z =   0.600 mm,
	W =180.000 deg,	P =   0.000 deg,	R =    90.000 deg
};
P[9312]{
   GP1:
	UF : 1, UT : 1,		CONFIG : 'N U T, 0, 0, 1',
	X =  82.000  mm,	Y =  202.000  mm,	Z =   15.000 mm,
	W =180.000 deg,	P =   0.000 deg,	R =    90.000 deg
};
P[9313]{
   GP1:
	UF : 1, UT : 1,		CONFIG : 'N U T, 0, 0, 1',
	X =  85.000  mm,	Y =  202.000  mm,	Z =   15.000 mm,
	W =180.000 deg,	P =   0.000 deg,	R =    90.000 deg
};
P[9314]{
   GP1:
	UF : 1, UT : 1,		CONFIG : 'N U T, 0, 0, 1',
	X =  85.000  mm,	Y =  202.000  mm,	Z =   0.600 mm,
	W =180.000 deg,	P =   0.000 deg,	R =    90.000 deg
};
P[9315]{
   GP1:
	UF : 1, UT : 1,		CONFIG : 'N U T, 0, 0, 1',
	X =  85.000  mm,	Y =  202.000  mm,	Z =   15.000 mm,
	W =180.000 deg,	P =   0.000 deg,	R =    90.000 deg
};
P[9316]{
   GP1:
	UF : 1, UT : 1,		CONFIG : 'N U T, 0, 0, 1',
	X =  88.000  mm,	Y =  202.000  mm,	Z =   15.000 mm,
	W =180.000 deg,	P =   0.000 deg,	R =    90.000 deg
};
P[9317]{
   GP1:
	UF : 1, UT : 1,		CONFIG : 'N U T, 0, 0, 1',
	X =  88.000  mm,	Y =  202.000  mm,	Z =   0.600 mm,
	W =180.000 deg,	P =   0.000 deg,	R =    90.000 deg
};
P[9318]{
   GP1:
	UF : 1, UT : 1,		CONFIG : 'N U T, 0, 0, 1',
	X =  88.000  mm,	Y =  202.000  mm,	Z =   15.000 mm,
	W =180.000 deg,	P =   0.000 deg,	R =    90.000 deg
};
P[9319]{
   GP1:
	UF : 1, UT : 1,		CONFIG : 'N U T, 0, 0, 1',
	X =  91.000  mm,	Y =  202.000  mm,	Z =   15.000 mm,
	W =180.000 deg,	P =   0.000 deg,	R =    90.000 deg
};
P[9320]{
   GP1:
	UF : 1, UT : 1,		CONFIG : 'N U T, 0, 0, 1',
	X =  91.000  mm,	Y =  202.000  mm,	Z =   0.600 mm,
	W =180.000 deg,	P =   0.000 deg,	R =    90.000 deg
};
P[9321]{
   GP1:
	UF : 1, UT : 1,		CONFIG : 'N U T, 0, 0, 1',
	X =  91.000  mm,	Y =  202.000  mm,	Z =   15.000 mm,
	W =180.000 deg,	P =   0.000 deg,	R =    90.000 deg
};
P[9322]{
   GP1:
	UF : 1, UT : 1,		CONFIG : 'N U T, 0, 0, 1',
	X =  94.000  mm,	Y =  202.000  mm,	Z =   15.000 mm,
	W =180.000 deg,	P =   0.000 deg,	R =    90.000 deg
};
P[9323]{
   GP1:
	UF : 1, UT : 1,		CONFIG : 'N U T, 0, 0, 1',
	X =  94.000  mm,	Y =  202.000  mm,	Z =   0.600 mm,
	W =180.000 deg,	P =   0.000 deg,	R =    90.000 deg
};
P[9324]{
   GP1:
	UF : 1, UT : 1,		CONFIG : 'N U T, 0, 0, 1',
	X =  94.000  mm,	Y =  202.000  mm,	Z =   15.000 mm,
	W =180.000 deg,	P =   0.000 deg,	R =    90.000 deg
};
P[9325]{
   GP1:
	UF : 1, UT : 1,		CONFIG : 'N U T, 0, 0, 1',
	X =  97.000  mm,	Y =  202.000  mm,	Z =   15.000 mm,
	W =180.000 deg,	P =   0.000 deg,	R =    90.000 deg
};
P[9326]{
   GP1:
	UF : 1, UT : 1,		CONFIG : 'N U T, 0, 0, 1',
	X =  97.000  mm,	Y =  202.000  mm,	Z =   0.600 mm,
	W =180.000 deg,	P =   0.000 deg,	R =    90.000 deg
};
P[9327]{
   GP1:
	UF : 1, UT : 1,		CONFIG : 'N U T, 0, 0, 1',
	X =  97.000  mm,	Y =  202.000  mm,	Z =   15.000 mm,
	W =180.000 deg,	P =   0.000 deg,	R =    90.000 deg
};
P[9328]{
   GP1:
	UF : 1, UT : 1,		CONFIG : 'N U T, 0, 0, 1',
	X =  100.000  mm,	Y =  202.000  mm,	Z =   15.000 mm,
	W =180.000 deg,	P =   0.000 deg,	R =    90.000 deg
};
P[9329]{
   GP1:
	UF : 1, UT : 1,		CONFIG : 'N U T, 0, 0, 1',
	X =  100.000  mm,	Y =  202.000  mm,	Z =   0.600 mm,
	W =180.000 deg,	P =   0.000 deg,	R =    90.000 deg
};
P[9330]{
   GP1:
	UF : 1, UT : 1,		CONFIG : 'N U T, 0, 0, 1',
	X =  100.000  mm,	Y =  202.000  mm,	Z =   15.000 mm,
	W =180.000 deg,	P =   0.000 deg,	R =    90.000 deg
};
P[9331]{
   GP1:
	UF : 1, UT : 1,		CONFIG : 'N U T, 0, 0, 1',
	X =  103.000  mm,	Y =  202.000  mm,	Z =   15.000 mm,
	W =180.000 deg,	P =   0.000 deg,	R =    90.000 deg
};
P[9332]{
   GP1:
	UF : 1, UT : 1,		CONFIG : 'N U T, 0, 0, 1',
	X =  103.000  mm,	Y =  202.000  mm,	Z =   0.600 mm,
	W =180.000 deg,	P =   0.000 deg,	R =    90.000 deg
};
P[9333]{
   GP1:
	UF : 1, UT : 1,		CONFIG : 'N U T, 0, 0, 1',
	X =  103.000  mm,	Y =  202.000  mm,	Z =   15.000 mm,
	W =180.000 deg,	P =   0.000 deg,	R =    90.000 deg
};
P[9334]{
   GP1:
	UF : 1, UT : 1,		CONFIG : 'N U T, 0, 0, 1',
	X =  106.000  mm,	Y =  202.000  mm,	Z =   15.000 mm,
	W =180.000 deg,	P =   0.000 deg,	R =    90.000 deg
};
P[9335]{
   GP1:
	UF : 1, UT : 1,		CONFIG : 'N U T, 0, 0, 1',
	X =  106.000  mm,	Y =  202.000  mm,	Z =   0.600 mm,
	W =180.000 deg,	P =   0.000 deg,	R =    90.000 deg
};
P[9336]{
   GP1:
	UF : 1, UT : 1,		CONFIG : 'N U T, 0, 0, 1',
	X =  106.000  mm,	Y =  202.000  mm,	Z =   15.000 mm,
	W =180.000 deg,	P =   0.000 deg,	R =    90.000 deg
};
P[9337]{
   GP1:
	UF : 1, UT : 1,		CONFIG : 'N U T, 0, 0, 1',
	X =  109.000  mm,	Y =  202.000  mm,	Z =   15.000 mm,
	W =180.000 deg,	P =   0.000 deg,	R =    90.000 deg
};
P[9338]{
   GP1:
	UF : 1, UT : 1,		CONFIG : 'N U T, 0, 0, 1',
	X =  109.000  mm,	Y =  202.000  mm,	Z =   0.600 mm,
	W =180.000 deg,	P =   0.000 deg,	R =    90.000 deg
};
P[9339]{
   GP1:
	UF : 1, UT : 1,		CONFIG : 'N U T, 0, 0, 1',
	X =  109.000  mm,	Y =  202.000  mm,	Z =   15.000 mm,
	W =180.000 deg,	P =   0.000 deg,	R =    90.000 deg
};
P[9340]{
   GP1:
	UF : 1, UT : 1,		CONFIG : 'N U T, 0, 0, 1',
	X =  112.000  mm,	Y =  202.000  mm,	Z =   15.000 mm,
	W =180.000 deg,	P =   0.000 deg,	R =    90.000 deg
};
P[9341]{
   GP1:
	UF : 1, UT : 1,		CONFIG : 'N U T, 0, 0, 1',
	X =  112.000  mm,	Y =  202.000  mm,	Z =   0.600 mm,
	W =180.000 deg,	P =   0.000 deg,	R =    90.000 deg
};
P[9342]{
   GP1:
	UF : 1, UT : 1,		CONFIG : 'N U T, 0, 0, 1',
	X =  112.000  mm,	Y =  202.000  mm,	Z =   15.000 mm,
	W =180.000 deg,	P =   0.000 deg,	R =    90.000 deg
};
P[9343]{
   GP1:
	UF : 1, UT : 1,		CONFIG : 'N U T, 0, 0, 1',
	X =  115.000  mm,	Y =  202.000  mm,	Z =   15.000 mm,
	W =180.000 deg,	P =   0.000 deg,	R =    90.000 deg
};
P[9344]{
   GP1:
	UF : 1, UT : 1,		CONFIG : 'N U T, 0, 0, 1',
	X =  115.000  mm,	Y =  202.000  mm,	Z =   0.600 mm,
	W =180.000 deg,	P =   0.000 deg,	R =    90.000 deg
};
P[9345]{
   GP1:
	UF : 1, UT : 1,		CONFIG : 'N U T, 0, 0, 1',
	X =  115.000  mm,	Y =  202.000  mm,	Z =   15.000 mm,
	W =180.000 deg,	P =   0.000 deg,	R =    90.000 deg
};
P[9346]{
   GP1:
	UF : 1, UT : 1,		CONFIG : 'N U T, 0, 0, 1',
	X =  118.000  mm,	Y =  202.000  mm,	Z =   15.000 mm,
	W =180.000 deg,	P =   0.000 deg,	R =    90.000 deg
};
P[9347]{
   GP1:
	UF : 1, UT : 1,		CONFIG : 'N U T, 0, 0, 1',
	X =  118.000  mm,	Y =  202.000  mm,	Z =   0.600 mm,
	W =180.000 deg,	P =   0.000 deg,	R =    90.000 deg
};
P[9348]{
   GP1:
	UF : 1, UT : 1,		CONFIG : 'N U T, 0, 0, 1',
	X =  118.000  mm,	Y =  202.000  mm,	Z =   15.000 mm,
	W =180.000 deg,	P =   0.000 deg,	R =    90.000 deg
};
P[9349]{
   GP1:
	UF : 1, UT : 1,		CONFIG : 'N U T, 0, 0, 1',
	X =  121.000  mm,	Y =  202.000  mm,	Z =   15.000 mm,
	W =180.000 deg,	P =   0.000 deg,	R =    90.000 deg
};
P[9350]{
   GP1:
	UF : 1, UT : 1,		CONFIG : 'N U T, 0, 0, 1',
	X =  121.000  mm,	Y =  202.000  mm,	Z =   0.600 mm,
	W =180.000 deg,	P =   0.000 deg,	R =    90.000 deg
};
P[9351]{
   GP1:
	UF : 1, UT : 1,		CONFIG : 'N U T, 0, 0, 1',
	X =  121.000  mm,	Y =  202.000  mm,	Z =   15.000 mm,
	W =180.000 deg,	P =   0.000 deg,	R =    90.000 deg
};
P[9352]{
   GP1:
	UF : 1, UT : 1,		CONFIG : 'N U T, 0, 0, 1',
	X =  124.000  mm,	Y =  202.000  mm,	Z =   15.000 mm,
	W =180.000 deg,	P =   0.000 deg,	R =    90.000 deg
};
P[9353]{
   GP1:
	UF : 1, UT : 1,		CONFIG : 'N U T, 0, 0, 1',
	X =  124.000  mm,	Y =  202.000  mm,	Z =   0.600 mm,
	W =180.000 deg,	P =   0.000 deg,	R =    90.000 deg
};
P[9354]{
   GP1:
	UF : 1, UT : 1,		CONFIG : 'N U T, 0, 0, 1',
	X =  124.000  mm,	Y =  202.000  mm,	Z =   15.000 mm,
	W =180.000 deg,	P =   0.000 deg,	R =    90.000 deg
};
P[9355]{
   GP1:
	UF : 1, UT : 1,		CONFIG : 'N U T, 0, 0, 1',
	X =  127.000  mm,	Y =  202.000  mm,	Z =   15.000 mm,
	W =180.000 deg,	P =   0.000 deg,	R =    90.000 deg
};
P[9356]{
   GP1:
	UF : 1, UT : 1,		CONFIG : 'N U T, 0, 0, 1',
	X =  127.000  mm,	Y =  202.000  mm,	Z =   0.600 mm,
	W =180.000 deg,	P =   0.000 deg,	R =    90.000 deg
};
P[9357]{
   GP1:
	UF : 1, UT : 1,		CONFIG : 'N U T, 0, 0, 1',
	X =  127.000  mm,	Y =  202.000  mm,	Z =   15.000 mm,
	W =180.000 deg,	P =   0.000 deg,	R =    90.000 deg
};
P[9358]{
   GP1:
	UF : 1, UT : 1,		CONFIG : 'N U T, 0, 0, 1',
	X =  130.000  mm,	Y =  202.000  mm,	Z =   15.000 mm,
	W =180.000 deg,	P =   0.000 deg,	R =    90.000 deg
};
P[9359]{
   GP1:
	UF : 1, UT : 1,		CONFIG : 'N U T, 0, 0, 1',
	X =  130.000  mm,	Y =  202.000  mm,	Z =   0.600 mm,
	W =180.000 deg,	P =   0.000 deg,	R =    90.000 deg
};
P[9360]{
   GP1:
	UF : 1, UT : 1,		CONFIG : 'N U T, 0, 0, 1',
	X =  130.000  mm,	Y =  202.000  mm,	Z =   15.000 mm,
	W =180.000 deg,	P =   0.000 deg,	R =    90.000 deg
};
P[9361]{
   GP1:
	UF : 1, UT : 1,		CONFIG : 'N U T, 0, 0, 1',
	X =  133.000  mm,	Y =  202.000  mm,	Z =   15.000 mm,
	W =180.000 deg,	P =   0.000 deg,	R =    90.000 deg
};
P[9362]{
   GP1:
	UF : 1, UT : 1,		CONFIG : 'N U T, 0, 0, 1',
	X =  133.000  mm,	Y =  202.000  mm,	Z =   0.600 mm,
	W =180.000 deg,	P =   0.000 deg,	R =    90.000 deg
};
P[9363]{
   GP1:
	UF : 1, UT : 1,		CONFIG : 'N U T, 0, 0, 1',
	X =  133.000  mm,	Y =  202.000  mm,	Z =   15.000 mm,
	W =180.000 deg,	P =   0.000 deg,	R =    90.000 deg
};
P[9364]{
   GP1:
	UF : 1, UT : 1,		CONFIG : 'N U T, 0, 0, 1',
	X =  136.000  mm,	Y =  202.000  mm,	Z =   15.000 mm,
	W =180.000 deg,	P =   0.000 deg,	R =    90.000 deg
};
P[9365]{
   GP1:
	UF : 1, UT : 1,		CONFIG : 'N U T, 0, 0, 1',
	X =  136.000  mm,	Y =  202.000  mm,	Z =   0.600 mm,
	W =180.000 deg,	P =   0.000 deg,	R =    90.000 deg
};
P[9366]{
   GP1:
	UF : 1, UT : 1,		CONFIG : 'N U T, 0, 0, 1',
	X =  136.000  mm,	Y =  202.000  mm,	Z =   15.000 mm,
	W =180.000 deg,	P =   0.000 deg,	R =    90.000 deg
};
P[9367]{
   GP1:
	UF : 1, UT : 1,		CONFIG : 'N U T, 0, 0, 1',
	X =  139.000  mm,	Y =  202.000  mm,	Z =   15.000 mm,
	W =180.000 deg,	P =   0.000 deg,	R =    90.000 deg
};
P[9368]{
   GP1:
	UF : 1, UT : 1,		CONFIG : 'N U T, 0, 0, 1',
	X =  139.000  mm,	Y =  202.000  mm,	Z =   0.600 mm,
	W =180.000 deg,	P =   0.000 deg,	R =    90.000 deg
};
P[9369]{
   GP1:
	UF : 1, UT : 1,		CONFIG : 'N U T, 0, 0, 1',
	X =  139.000  mm,	Y =  202.000  mm,	Z =   15.000 mm,
	W =180.000 deg,	P =   0.000 deg,	R =    90.000 deg
};
P[9370]{
   GP1:
	UF : 1, UT : 1,		CONFIG : 'N U T, 0, 0, 1',
	X =  142.000  mm,	Y =  202.000  mm,	Z =   15.000 mm,
	W =180.000 deg,	P =   0.000 deg,	R =    90.000 deg
};
P[9371]{
   GP1:
	UF : 1, UT : 1,		CONFIG : 'N U T, 0, 0, 1',
	X =  142.000  mm,	Y =  202.000  mm,	Z =   0.600 mm,
	W =180.000 deg,	P =   0.000 deg,	R =    90.000 deg
};
P[9372]{
   GP1:
	UF : 1, UT : 1,		CONFIG : 'N U T, 0, 0, 1',
	X =  142.000  mm,	Y =  202.000  mm,	Z =   15.000 mm,
	W =180.000 deg,	P =   0.000 deg,	R =    90.000 deg
};
P[9373]{
   GP1:
	UF : 1, UT : 1,		CONFIG : 'N U T, 0, 0, 1',
	X =  145.000  mm,	Y =  202.000  mm,	Z =   15.000 mm,
	W =180.000 deg,	P =   0.000 deg,	R =    90.000 deg
};
P[9374]{
   GP1:
	UF : 1, UT : 1,		CONFIG : 'N U T, 0, 0, 1',
	X =  145.000  mm,	Y =  202.000  mm,	Z =   0.600 mm,
	W =180.000 deg,	P =   0.000 deg,	R =    90.000 deg
};
P[9375]{
   GP1:
	UF : 1, UT : 1,		CONFIG : 'N U T, 0, 0, 1',
	X =  145.000  mm,	Y =  202.000  mm,	Z =   15.000 mm,
	W =180.000 deg,	P =   0.000 deg,	R =    90.000 deg
};
P[9376]{
   GP1:
	UF : 1, UT : 1,		CONFIG : 'N U T, 0, 0, 1',
	X =  148.000  mm,	Y =  202.000  mm,	Z =   15.000 mm,
	W =180.000 deg,	P =   0.000 deg,	R =    90.000 deg
};
P[9377]{
   GP1:
	UF : 1, UT : 1,		CONFIG : 'N U T, 0, 0, 1',
	X =  148.000  mm,	Y =  202.000  mm,	Z =   0.600 mm,
	W =180.000 deg,	P =   0.000 deg,	R =    90.000 deg
};
P[9378]{
   GP1:
	UF : 1, UT : 1,		CONFIG : 'N U T, 0, 0, 1',
	X =  148.000  mm,	Y =  202.000  mm,	Z =   15.000 mm,
	W =180.000 deg,	P =   0.000 deg,	R =    90.000 deg
};
P[9379]{
   GP1:
	UF : 1, UT : 1,		CONFIG : 'N U T, 0, 0, 1',
	X =  151.000  mm,	Y =  202.000  mm,	Z =   15.000 mm,
	W =180.000 deg,	P =   0.000 deg,	R =    90.000 deg
};
P[9380]{
   GP1:
	UF : 1, UT : 1,		CONFIG : 'N U T, 0, 0, 1',
	X =  151.000  mm,	Y =  202.000  mm,	Z =   0.600 mm,
	W =180.000 deg,	P =   0.000 deg,	R =    90.000 deg
};
P[9381]{
   GP1:
	UF : 1, UT : 1,		CONFIG : 'N U T, 0, 0, 1',
	X =  151.000  mm,	Y =  202.000  mm,	Z =   15.000 mm,
	W =180.000 deg,	P =   0.000 deg,	R =    90.000 deg
};
P[9382]{
   GP1:
	UF : 1, UT : 1,		CONFIG : 'N U T, 0, 0, 1',
	X =  154.000  mm,	Y =  202.000  mm,	Z =   15.000 mm,
	W =180.000 deg,	P =   0.000 deg,	R =    90.000 deg
};
P[9383]{
   GP1:
	UF : 1, UT : 1,		CONFIG : 'N U T, 0, 0, 1',
	X =  154.000  mm,	Y =  202.000  mm,	Z =   0.600 mm,
	W =180.000 deg,	P =   0.000 deg,	R =    90.000 deg
};
P[9384]{
   GP1:
	UF : 1, UT : 1,		CONFIG : 'N U T, 0, 0, 1',
	X =  154.000  mm,	Y =  202.000  mm,	Z =   15.000 mm,
	W =180.000 deg,	P =   0.000 deg,	R =    90.000 deg
};
P[9385]{
   GP1:
	UF : 1, UT : 1,		CONFIG : 'N U T, 0, 0, 1',
	X =  157.000  mm,	Y =  202.000  mm,	Z =   15.000 mm,
	W =180.000 deg,	P =   0.000 deg,	R =    90.000 deg
};
P[9386]{
   GP1:
	UF : 1, UT : 1,		CONFIG : 'N U T, 0, 0, 1',
	X =  157.000  mm,	Y =  202.000  mm,	Z =   0.600 mm,
	W =180.000 deg,	P =   0.000 deg,	R =    90.000 deg
};
P[9387]{
   GP1:
	UF : 1, UT : 1,		CONFIG : 'N U T, 0, 0, 1',
	X =  157.000  mm,	Y =  202.000  mm,	Z =   15.000 mm,
	W =180.000 deg,	P =   0.000 deg,	R =    90.000 deg
};
P[9388]{
   GP1:
	UF : 1, UT : 1,		CONFIG : 'N U T, 0, 0, 1',
	X =  160.000  mm,	Y =  202.000  mm,	Z =   15.000 mm,
	W =180.000 deg,	P =   0.000 deg,	R =    90.000 deg
};
P[9389]{
   GP1:
	UF : 1, UT : 1,		CONFIG : 'N U T, 0, 0, 1',
	X =  160.000  mm,	Y =  202.000  mm,	Z =   0.600 mm,
	W =180.000 deg,	P =   0.000 deg,	R =    90.000 deg
};
P[9390]{
   GP1:
	UF : 1, UT : 1,		CONFIG : 'N U T, 0, 0, 1',
	X =  160.000  mm,	Y =  202.000  mm,	Z =   15.000 mm,
	W =180.000 deg,	P =   0.000 deg,	R =    90.000 deg
};
P[9391]{
   GP1:
	UF : 1, UT : 1,		CONFIG : 'N U T, 0, 0, 1',
	X =  163.000  mm,	Y =  202.000  mm,	Z =   15.000 mm,
	W =180.000 deg,	P =   0.000 deg,	R =    90.000 deg
};
P[9392]{
   GP1:
	UF : 1, UT : 1,		CONFIG : 'N U T, 0, 0, 1',
	X =  163.000  mm,	Y =  202.000  mm,	Z =   0.600 mm,
	W =180.000 deg,	P =   0.000 deg,	R =    90.000 deg
};
P[9393]{
   GP1:
	UF : 1, UT : 1,		CONFIG : 'N U T, 0, 0, 1',
	X =  163.000  mm,	Y =  202.000  mm,	Z =   15.000 mm,
	W =180.000 deg,	P =   0.000 deg,	R =    90.000 deg
};
P[9394]{
   GP1:
	UF : 1, UT : 1,		CONFIG : 'N U T, 0, 0, 1',
	X =  166.000  mm,	Y =  202.000  mm,	Z =   15.000 mm,
	W =180.000 deg,	P =   0.000 deg,	R =    90.000 deg
};
P[9395]{
   GP1:
	UF : 1, UT : 1,		CONFIG : 'N U T, 0, 0, 1',
	X =  166.000  mm,	Y =  202.000  mm,	Z =   0.600 mm,
	W =180.000 deg,	P =   0.000 deg,	R =    90.000 deg
};
P[9396]{
   GP1:
	UF : 1, UT : 1,		CONFIG : 'N U T, 0, 0, 1',
	X =  166.000  mm,	Y =  202.000  mm,	Z =   15.000 mm,
	W =180.000 deg,	P =   0.000 deg,	R =    90.000 deg
};
P[9397]{
   GP1:
	UF : 1, UT : 1,		CONFIG : 'N U T, 0, 0, 1',
	X =  169.000  mm,	Y =  202.000  mm,	Z =   15.000 mm,
	W =180.000 deg,	P =   0.000 deg,	R =    90.000 deg
};
P[9398]{
   GP1:
	UF : 1, UT : 1,		CONFIG : 'N U T, 0, 0, 1',
	X =  169.000  mm,	Y =  202.000  mm,	Z =   0.600 mm,
	W =180.000 deg,	P =   0.000 deg,	R =    90.000 deg
};
P[9399]{
   GP1:
	UF : 1, UT : 1,		CONFIG : 'N U T, 0, 0, 1',
	X =  169.000  mm,	Y =  202.000  mm,	Z =   15.000 mm,
	W =180.000 deg,	P =   0.000 deg,	R =    90.000 deg
};
P[9400]{
   GP1:
	UF : 1, UT : 1,		CONFIG : 'N U T, 0, 0, 1',
	X =  172.000  mm,	Y =  202.000  mm,	Z =   15.000 mm,
	W =180.000 deg,	P =   0.000 deg,	R =    90.000 deg
};
P[9401]{
   GP1:
	UF : 1, UT : 1,		CONFIG : 'N U T, 0, 0, 1',
	X =  172.000  mm,	Y =  202.000  mm,	Z =   0.600 mm,
	W =180.000 deg,	P =   0.000 deg,	R =    90.000 deg
};
P[9402]{
   GP1:
	UF : 1, UT : 1,		CONFIG : 'N U T, 0, 0, 1',
	X =  172.000  mm,	Y =  202.000  mm,	Z =   15.000 mm,
	W =180.000 deg,	P =   0.000 deg,	R =    90.000 deg
};
P[9403]{
   GP1:
	UF : 1, UT : 1,		CONFIG : 'N U T, 0, 0, 1',
	X =  175.000  mm,	Y =  202.000  mm,	Z =   15.000 mm,
	W =180.000 deg,	P =   0.000 deg,	R =    90.000 deg
};
P[9404]{
   GP1:
	UF : 1, UT : 1,		CONFIG : 'N U T, 0, 0, 1',
	X =  175.000  mm,	Y =  202.000  mm,	Z =   0.600 mm,
	W =180.000 deg,	P =   0.000 deg,	R =    90.000 deg
};
P[9405]{
   GP1:
	UF : 1, UT : 1,		CONFIG : 'N U T, 0, 0, 1',
	X =  175.000  mm,	Y =  202.000  mm,	Z =   15.000 mm,
	W =180.000 deg,	P =   0.000 deg,	R =    90.000 deg
};
P[9406]{
   GP1:
	UF : 1, UT : 1,		CONFIG : 'N U T, 0, 0, 1',
	X =  178.000  mm,	Y =  202.000  mm,	Z =   15.000 mm,
	W =180.000 deg,	P =   0.000 deg,	R =    90.000 deg
};
P[9407]{
   GP1:
	UF : 1, UT : 1,		CONFIG : 'N U T, 0, 0, 1',
	X =  178.000  mm,	Y =  202.000  mm,	Z =   0.600 mm,
	W =180.000 deg,	P =   0.000 deg,	R =    90.000 deg
};
P[9408]{
   GP1:
	UF : 1, UT : 1,		CONFIG : 'N U T, 0, 0, 1',
	X =  178.000  mm,	Y =  202.000  mm,	Z =   15.000 mm,
	W =180.000 deg,	P =   0.000 deg,	R =    90.000 deg
};
P[9409]{
   GP1:
	UF : 1, UT : 1,		CONFIG : 'N U T, 0, 0, 1',
	X =  1.000  mm,	Y =  205.000  mm,	Z =   15.000 mm,
	W =180.000 deg,	P =   0.000 deg,	R =    90.000 deg
};
P[9410]{
   GP1:
	UF : 1, UT : 1,		CONFIG : 'N U T, 0, 0, 1',
	X =  1.000  mm,	Y =  205.000  mm,	Z =   0.600 mm,
	W =180.000 deg,	P =   0.000 deg,	R =    90.000 deg
};
P[9411]{
   GP1:
	UF : 1, UT : 1,		CONFIG : 'N U T, 0, 0, 1',
	X =  1.000  mm,	Y =  205.000  mm,	Z =   15.000 mm,
	W =180.000 deg,	P =   0.000 deg,	R =    90.000 deg
};
P[9412]{
   GP1:
	UF : 1, UT : 1,		CONFIG : 'N U T, 0, 0, 1',
	X =  4.000  mm,	Y =  205.000  mm,	Z =   15.000 mm,
	W =180.000 deg,	P =   0.000 deg,	R =    90.000 deg
};
P[9413]{
   GP1:
	UF : 1, UT : 1,		CONFIG : 'N U T, 0, 0, 1',
	X =  4.000  mm,	Y =  205.000  mm,	Z =   0.600 mm,
	W =180.000 deg,	P =   0.000 deg,	R =    90.000 deg
};
P[9414]{
   GP1:
	UF : 1, UT : 1,		CONFIG : 'N U T, 0, 0, 1',
	X =  4.000  mm,	Y =  205.000  mm,	Z =   15.000 mm,
	W =180.000 deg,	P =   0.000 deg,	R =    90.000 deg
};
P[9415]{
   GP1:
	UF : 1, UT : 1,		CONFIG : 'N U T, 0, 0, 1',
	X =  7.000  mm,	Y =  205.000  mm,	Z =   15.000 mm,
	W =180.000 deg,	P =   0.000 deg,	R =    90.000 deg
};
P[9416]{
   GP1:
	UF : 1, UT : 1,		CONFIG : 'N U T, 0, 0, 1',
	X =  7.000  mm,	Y =  205.000  mm,	Z =   0.600 mm,
	W =180.000 deg,	P =   0.000 deg,	R =    90.000 deg
};
P[9417]{
   GP1:
	UF : 1, UT : 1,		CONFIG : 'N U T, 0, 0, 1',
	X =  7.000  mm,	Y =  205.000  mm,	Z =   15.000 mm,
	W =180.000 deg,	P =   0.000 deg,	R =    90.000 deg
};
P[9418]{
   GP1:
	UF : 1, UT : 1,		CONFIG : 'N U T, 0, 0, 1',
	X =  10.000  mm,	Y =  205.000  mm,	Z =   15.000 mm,
	W =180.000 deg,	P =   0.000 deg,	R =    90.000 deg
};
P[9419]{
   GP1:
	UF : 1, UT : 1,		CONFIG : 'N U T, 0, 0, 1',
	X =  10.000  mm,	Y =  205.000  mm,	Z =   0.600 mm,
	W =180.000 deg,	P =   0.000 deg,	R =    90.000 deg
};
P[9420]{
   GP1:
	UF : 1, UT : 1,		CONFIG : 'N U T, 0, 0, 1',
	X =  10.000  mm,	Y =  205.000  mm,	Z =   15.000 mm,
	W =180.000 deg,	P =   0.000 deg,	R =    90.000 deg
};
P[9421]{
   GP1:
	UF : 1, UT : 1,		CONFIG : 'N U T, 0, 0, 1',
	X =  13.000  mm,	Y =  205.000  mm,	Z =   15.000 mm,
	W =180.000 deg,	P =   0.000 deg,	R =    90.000 deg
};
P[9422]{
   GP1:
	UF : 1, UT : 1,		CONFIG : 'N U T, 0, 0, 1',
	X =  13.000  mm,	Y =  205.000  mm,	Z =   0.600 mm,
	W =180.000 deg,	P =   0.000 deg,	R =    90.000 deg
};
P[9423]{
   GP1:
	UF : 1, UT : 1,		CONFIG : 'N U T, 0, 0, 1',
	X =  13.000  mm,	Y =  205.000  mm,	Z =   15.000 mm,
	W =180.000 deg,	P =   0.000 deg,	R =    90.000 deg
};
P[9424]{
   GP1:
	UF : 1, UT : 1,		CONFIG : 'N U T, 0, 0, 1',
	X =  16.000  mm,	Y =  205.000  mm,	Z =   15.000 mm,
	W =180.000 deg,	P =   0.000 deg,	R =    90.000 deg
};
P[9425]{
   GP1:
	UF : 1, UT : 1,		CONFIG : 'N U T, 0, 0, 1',
	X =  16.000  mm,	Y =  205.000  mm,	Z =   0.600 mm,
	W =180.000 deg,	P =   0.000 deg,	R =    90.000 deg
};
P[9426]{
   GP1:
	UF : 1, UT : 1,		CONFIG : 'N U T, 0, 0, 1',
	X =  16.000  mm,	Y =  205.000  mm,	Z =   15.000 mm,
	W =180.000 deg,	P =   0.000 deg,	R =    90.000 deg
};
P[9427]{
   GP1:
	UF : 1, UT : 1,		CONFIG : 'N U T, 0, 0, 1',
	X =  19.000  mm,	Y =  205.000  mm,	Z =   15.000 mm,
	W =180.000 deg,	P =   0.000 deg,	R =    90.000 deg
};
P[9428]{
   GP1:
	UF : 1, UT : 1,		CONFIG : 'N U T, 0, 0, 1',
	X =  19.000  mm,	Y =  205.000  mm,	Z =   0.600 mm,
	W =180.000 deg,	P =   0.000 deg,	R =    90.000 deg
};
P[9429]{
   GP1:
	UF : 1, UT : 1,		CONFIG : 'N U T, 0, 0, 1',
	X =  19.000  mm,	Y =  205.000  mm,	Z =   15.000 mm,
	W =180.000 deg,	P =   0.000 deg,	R =    90.000 deg
};
P[9430]{
   GP1:
	UF : 1, UT : 1,		CONFIG : 'N U T, 0, 0, 1',
	X =  22.000  mm,	Y =  205.000  mm,	Z =   15.000 mm,
	W =180.000 deg,	P =   0.000 deg,	R =    90.000 deg
};
P[9431]{
   GP1:
	UF : 1, UT : 1,		CONFIG : 'N U T, 0, 0, 1',
	X =  22.000  mm,	Y =  205.000  mm,	Z =   0.600 mm,
	W =180.000 deg,	P =   0.000 deg,	R =    90.000 deg
};
P[9432]{
   GP1:
	UF : 1, UT : 1,		CONFIG : 'N U T, 0, 0, 1',
	X =  22.000  mm,	Y =  205.000  mm,	Z =   15.000 mm,
	W =180.000 deg,	P =   0.000 deg,	R =    90.000 deg
};
P[9433]{
   GP1:
	UF : 1, UT : 1,		CONFIG : 'N U T, 0, 0, 1',
	X =  25.000  mm,	Y =  205.000  mm,	Z =   15.000 mm,
	W =180.000 deg,	P =   0.000 deg,	R =    90.000 deg
};
P[9434]{
   GP1:
	UF : 1, UT : 1,		CONFIG : 'N U T, 0, 0, 1',
	X =  25.000  mm,	Y =  205.000  mm,	Z =   0.600 mm,
	W =180.000 deg,	P =   0.000 deg,	R =    90.000 deg
};
P[9435]{
   GP1:
	UF : 1, UT : 1,		CONFIG : 'N U T, 0, 0, 1',
	X =  25.000  mm,	Y =  205.000  mm,	Z =   15.000 mm,
	W =180.000 deg,	P =   0.000 deg,	R =    90.000 deg
};
P[9436]{
   GP1:
	UF : 1, UT : 1,		CONFIG : 'N U T, 0, 0, 1',
	X =  28.000  mm,	Y =  205.000  mm,	Z =   15.000 mm,
	W =180.000 deg,	P =   0.000 deg,	R =    90.000 deg
};
P[9437]{
   GP1:
	UF : 1, UT : 1,		CONFIG : 'N U T, 0, 0, 1',
	X =  28.000  mm,	Y =  205.000  mm,	Z =   0.600 mm,
	W =180.000 deg,	P =   0.000 deg,	R =    90.000 deg
};
P[9438]{
   GP1:
	UF : 1, UT : 1,		CONFIG : 'N U T, 0, 0, 1',
	X =  28.000  mm,	Y =  205.000  mm,	Z =   15.000 mm,
	W =180.000 deg,	P =   0.000 deg,	R =    90.000 deg
};
P[9439]{
   GP1:
	UF : 1, UT : 1,		CONFIG : 'N U T, 0, 0, 1',
	X =  31.000  mm,	Y =  205.000  mm,	Z =   15.000 mm,
	W =180.000 deg,	P =   0.000 deg,	R =    90.000 deg
};
P[9440]{
   GP1:
	UF : 1, UT : 1,		CONFIG : 'N U T, 0, 0, 1',
	X =  31.000  mm,	Y =  205.000  mm,	Z =   0.600 mm,
	W =180.000 deg,	P =   0.000 deg,	R =    90.000 deg
};
P[9441]{
   GP1:
	UF : 1, UT : 1,		CONFIG : 'N U T, 0, 0, 1',
	X =  31.000  mm,	Y =  205.000  mm,	Z =   15.000 mm,
	W =180.000 deg,	P =   0.000 deg,	R =    90.000 deg
};
P[9442]{
   GP1:
	UF : 1, UT : 1,		CONFIG : 'N U T, 0, 0, 1',
	X =  34.000  mm,	Y =  205.000  mm,	Z =   15.000 mm,
	W =180.000 deg,	P =   0.000 deg,	R =    90.000 deg
};
P[9443]{
   GP1:
	UF : 1, UT : 1,		CONFIG : 'N U T, 0, 0, 1',
	X =  34.000  mm,	Y =  205.000  mm,	Z =   0.600 mm,
	W =180.000 deg,	P =   0.000 deg,	R =    90.000 deg
};
P[9444]{
   GP1:
	UF : 1, UT : 1,		CONFIG : 'N U T, 0, 0, 1',
	X =  34.000  mm,	Y =  205.000  mm,	Z =   15.000 mm,
	W =180.000 deg,	P =   0.000 deg,	R =    90.000 deg
};
P[9445]{
   GP1:
	UF : 1, UT : 1,		CONFIG : 'N U T, 0, 0, 1',
	X =  37.000  mm,	Y =  205.000  mm,	Z =   15.000 mm,
	W =180.000 deg,	P =   0.000 deg,	R =    90.000 deg
};
P[9446]{
   GP1:
	UF : 1, UT : 1,		CONFIG : 'N U T, 0, 0, 1',
	X =  37.000  mm,	Y =  205.000  mm,	Z =   0.600 mm,
	W =180.000 deg,	P =   0.000 deg,	R =    90.000 deg
};
P[9447]{
   GP1:
	UF : 1, UT : 1,		CONFIG : 'N U T, 0, 0, 1',
	X =  37.000  mm,	Y =  205.000  mm,	Z =   15.000 mm,
	W =180.000 deg,	P =   0.000 deg,	R =    90.000 deg
};
P[9448]{
   GP1:
	UF : 1, UT : 1,		CONFIG : 'N U T, 0, 0, 1',
	X =  40.000  mm,	Y =  205.000  mm,	Z =   15.000 mm,
	W =180.000 deg,	P =   0.000 deg,	R =    90.000 deg
};
P[9449]{
   GP1:
	UF : 1, UT : 1,		CONFIG : 'N U T, 0, 0, 1',
	X =  40.000  mm,	Y =  205.000  mm,	Z =   0.600 mm,
	W =180.000 deg,	P =   0.000 deg,	R =    90.000 deg
};
P[9450]{
   GP1:
	UF : 1, UT : 1,		CONFIG : 'N U T, 0, 0, 1',
	X =  40.000  mm,	Y =  205.000  mm,	Z =   15.000 mm,
	W =180.000 deg,	P =   0.000 deg,	R =    90.000 deg
};
P[9451]{
   GP1:
	UF : 1, UT : 1,		CONFIG : 'N U T, 0, 0, 1',
	X =  43.000  mm,	Y =  205.000  mm,	Z =   15.000 mm,
	W =180.000 deg,	P =   0.000 deg,	R =    90.000 deg
};
P[9452]{
   GP1:
	UF : 1, UT : 1,		CONFIG : 'N U T, 0, 0, 1',
	X =  43.000  mm,	Y =  205.000  mm,	Z =   0.600 mm,
	W =180.000 deg,	P =   0.000 deg,	R =    90.000 deg
};
P[9453]{
   GP1:
	UF : 1, UT : 1,		CONFIG : 'N U T, 0, 0, 1',
	X =  43.000  mm,	Y =  205.000  mm,	Z =   15.000 mm,
	W =180.000 deg,	P =   0.000 deg,	R =    90.000 deg
};
P[9454]{
   GP1:
	UF : 1, UT : 1,		CONFIG : 'N U T, 0, 0, 1',
	X =  46.000  mm,	Y =  205.000  mm,	Z =   15.000 mm,
	W =180.000 deg,	P =   0.000 deg,	R =    90.000 deg
};
P[9455]{
   GP1:
	UF : 1, UT : 1,		CONFIG : 'N U T, 0, 0, 1',
	X =  46.000  mm,	Y =  205.000  mm,	Z =   0.600 mm,
	W =180.000 deg,	P =   0.000 deg,	R =    90.000 deg
};
P[9456]{
   GP1:
	UF : 1, UT : 1,		CONFIG : 'N U T, 0, 0, 1',
	X =  46.000  mm,	Y =  205.000  mm,	Z =   15.000 mm,
	W =180.000 deg,	P =   0.000 deg,	R =    90.000 deg
};
P[9457]{
   GP1:
	UF : 1, UT : 1,		CONFIG : 'N U T, 0, 0, 1',
	X =  49.000  mm,	Y =  205.000  mm,	Z =   15.000 mm,
	W =180.000 deg,	P =   0.000 deg,	R =    90.000 deg
};
P[9458]{
   GP1:
	UF : 1, UT : 1,		CONFIG : 'N U T, 0, 0, 1',
	X =  49.000  mm,	Y =  205.000  mm,	Z =   0.600 mm,
	W =180.000 deg,	P =   0.000 deg,	R =    90.000 deg
};
P[9459]{
   GP1:
	UF : 1, UT : 1,		CONFIG : 'N U T, 0, 0, 1',
	X =  49.000  mm,	Y =  205.000  mm,	Z =   15.000 mm,
	W =180.000 deg,	P =   0.000 deg,	R =    90.000 deg
};
P[9460]{
   GP1:
	UF : 1, UT : 1,		CONFIG : 'N U T, 0, 0, 1',
	X =  52.000  mm,	Y =  205.000  mm,	Z =   15.000 mm,
	W =180.000 deg,	P =   0.000 deg,	R =    90.000 deg
};
P[9461]{
   GP1:
	UF : 1, UT : 1,		CONFIG : 'N U T, 0, 0, 1',
	X =  52.000  mm,	Y =  205.000  mm,	Z =   0.600 mm,
	W =180.000 deg,	P =   0.000 deg,	R =    90.000 deg
};
P[9462]{
   GP1:
	UF : 1, UT : 1,		CONFIG : 'N U T, 0, 0, 1',
	X =  52.000  mm,	Y =  205.000  mm,	Z =   15.000 mm,
	W =180.000 deg,	P =   0.000 deg,	R =    90.000 deg
};
P[9463]{
   GP1:
	UF : 1, UT : 1,		CONFIG : 'N U T, 0, 0, 1',
	X =  55.000  mm,	Y =  205.000  mm,	Z =   15.000 mm,
	W =180.000 deg,	P =   0.000 deg,	R =    90.000 deg
};
P[9464]{
   GP1:
	UF : 1, UT : 1,		CONFIG : 'N U T, 0, 0, 1',
	X =  55.000  mm,	Y =  205.000  mm,	Z =   0.600 mm,
	W =180.000 deg,	P =   0.000 deg,	R =    90.000 deg
};
P[9465]{
   GP1:
	UF : 1, UT : 1,		CONFIG : 'N U T, 0, 0, 1',
	X =  55.000  mm,	Y =  205.000  mm,	Z =   15.000 mm,
	W =180.000 deg,	P =   0.000 deg,	R =    90.000 deg
};
P[9466]{
   GP1:
	UF : 1, UT : 1,		CONFIG : 'N U T, 0, 0, 1',
	X =  58.000  mm,	Y =  205.000  mm,	Z =   15.000 mm,
	W =180.000 deg,	P =   0.000 deg,	R =    90.000 deg
};
P[9467]{
   GP1:
	UF : 1, UT : 1,		CONFIG : 'N U T, 0, 0, 1',
	X =  58.000  mm,	Y =  205.000  mm,	Z =   0.600 mm,
	W =180.000 deg,	P =   0.000 deg,	R =    90.000 deg
};
P[9468]{
   GP1:
	UF : 1, UT : 1,		CONFIG : 'N U T, 0, 0, 1',
	X =  58.000  mm,	Y =  205.000  mm,	Z =   15.000 mm,
	W =180.000 deg,	P =   0.000 deg,	R =    90.000 deg
};
P[9469]{
   GP1:
	UF : 1, UT : 1,		CONFIG : 'N U T, 0, 0, 1',
	X =  61.000  mm,	Y =  205.000  mm,	Z =   15.000 mm,
	W =180.000 deg,	P =   0.000 deg,	R =    90.000 deg
};
P[9470]{
   GP1:
	UF : 1, UT : 1,		CONFIG : 'N U T, 0, 0, 1',
	X =  61.000  mm,	Y =  205.000  mm,	Z =   0.600 mm,
	W =180.000 deg,	P =   0.000 deg,	R =    90.000 deg
};
P[9471]{
   GP1:
	UF : 1, UT : 1,		CONFIG : 'N U T, 0, 0, 1',
	X =  61.000  mm,	Y =  205.000  mm,	Z =   15.000 mm,
	W =180.000 deg,	P =   0.000 deg,	R =    90.000 deg
};
P[9472]{
   GP1:
	UF : 1, UT : 1,		CONFIG : 'N U T, 0, 0, 1',
	X =  64.000  mm,	Y =  205.000  mm,	Z =   15.000 mm,
	W =180.000 deg,	P =   0.000 deg,	R =    90.000 deg
};
P[9473]{
   GP1:
	UF : 1, UT : 1,		CONFIG : 'N U T, 0, 0, 1',
	X =  64.000  mm,	Y =  205.000  mm,	Z =   0.600 mm,
	W =180.000 deg,	P =   0.000 deg,	R =    90.000 deg
};
P[9474]{
   GP1:
	UF : 1, UT : 1,		CONFIG : 'N U T, 0, 0, 1',
	X =  64.000  mm,	Y =  205.000  mm,	Z =   15.000 mm,
	W =180.000 deg,	P =   0.000 deg,	R =    90.000 deg
};
P[9475]{
   GP1:
	UF : 1, UT : 1,		CONFIG : 'N U T, 0, 0, 1',
	X =  67.000  mm,	Y =  205.000  mm,	Z =   15.000 mm,
	W =180.000 deg,	P =   0.000 deg,	R =    90.000 deg
};
P[9476]{
   GP1:
	UF : 1, UT : 1,		CONFIG : 'N U T, 0, 0, 1',
	X =  67.000  mm,	Y =  205.000  mm,	Z =   0.600 mm,
	W =180.000 deg,	P =   0.000 deg,	R =    90.000 deg
};
P[9477]{
   GP1:
	UF : 1, UT : 1,		CONFIG : 'N U T, 0, 0, 1',
	X =  67.000  mm,	Y =  205.000  mm,	Z =   15.000 mm,
	W =180.000 deg,	P =   0.000 deg,	R =    90.000 deg
};
P[9478]{
   GP1:
	UF : 1, UT : 1,		CONFIG : 'N U T, 0, 0, 1',
	X =  70.000  mm,	Y =  205.000  mm,	Z =   15.000 mm,
	W =180.000 deg,	P =   0.000 deg,	R =    90.000 deg
};
P[9479]{
   GP1:
	UF : 1, UT : 1,		CONFIG : 'N U T, 0, 0, 1',
	X =  70.000  mm,	Y =  205.000  mm,	Z =   0.600 mm,
	W =180.000 deg,	P =   0.000 deg,	R =    90.000 deg
};
P[9480]{
   GP1:
	UF : 1, UT : 1,		CONFIG : 'N U T, 0, 0, 1',
	X =  70.000  mm,	Y =  205.000  mm,	Z =   15.000 mm,
	W =180.000 deg,	P =   0.000 deg,	R =    90.000 deg
};
P[9481]{
   GP1:
	UF : 1, UT : 1,		CONFIG : 'N U T, 0, 0, 1',
	X =  73.000  mm,	Y =  205.000  mm,	Z =   15.000 mm,
	W =180.000 deg,	P =   0.000 deg,	R =    90.000 deg
};
P[9482]{
   GP1:
	UF : 1, UT : 1,		CONFIG : 'N U T, 0, 0, 1',
	X =  73.000  mm,	Y =  205.000  mm,	Z =   0.600 mm,
	W =180.000 deg,	P =   0.000 deg,	R =    90.000 deg
};
P[9483]{
   GP1:
	UF : 1, UT : 1,		CONFIG : 'N U T, 0, 0, 1',
	X =  73.000  mm,	Y =  205.000  mm,	Z =   15.000 mm,
	W =180.000 deg,	P =   0.000 deg,	R =    90.000 deg
};
P[9484]{
   GP1:
	UF : 1, UT : 1,		CONFIG : 'N U T, 0, 0, 1',
	X =  76.000  mm,	Y =  205.000  mm,	Z =   15.000 mm,
	W =180.000 deg,	P =   0.000 deg,	R =    90.000 deg
};
P[9485]{
   GP1:
	UF : 1, UT : 1,		CONFIG : 'N U T, 0, 0, 1',
	X =  76.000  mm,	Y =  205.000  mm,	Z =   0.600 mm,
	W =180.000 deg,	P =   0.000 deg,	R =    90.000 deg
};
P[9486]{
   GP1:
	UF : 1, UT : 1,		CONFIG : 'N U T, 0, 0, 1',
	X =  76.000  mm,	Y =  205.000  mm,	Z =   15.000 mm,
	W =180.000 deg,	P =   0.000 deg,	R =    90.000 deg
};
P[9487]{
   GP1:
	UF : 1, UT : 1,		CONFIG : 'N U T, 0, 0, 1',
	X =  79.000  mm,	Y =  205.000  mm,	Z =   15.000 mm,
	W =180.000 deg,	P =   0.000 deg,	R =    90.000 deg
};
P[9488]{
   GP1:
	UF : 1, UT : 1,		CONFIG : 'N U T, 0, 0, 1',
	X =  79.000  mm,	Y =  205.000  mm,	Z =   0.600 mm,
	W =180.000 deg,	P =   0.000 deg,	R =    90.000 deg
};
P[9489]{
   GP1:
	UF : 1, UT : 1,		CONFIG : 'N U T, 0, 0, 1',
	X =  79.000  mm,	Y =  205.000  mm,	Z =   15.000 mm,
	W =180.000 deg,	P =   0.000 deg,	R =    90.000 deg
};
P[9490]{
   GP1:
	UF : 1, UT : 1,		CONFIG : 'N U T, 0, 0, 1',
	X =  82.000  mm,	Y =  205.000  mm,	Z =   15.000 mm,
	W =180.000 deg,	P =   0.000 deg,	R =    90.000 deg
};
P[9491]{
   GP1:
	UF : 1, UT : 1,		CONFIG : 'N U T, 0, 0, 1',
	X =  82.000  mm,	Y =  205.000  mm,	Z =   0.600 mm,
	W =180.000 deg,	P =   0.000 deg,	R =    90.000 deg
};
P[9492]{
   GP1:
	UF : 1, UT : 1,		CONFIG : 'N U T, 0, 0, 1',
	X =  82.000  mm,	Y =  205.000  mm,	Z =   15.000 mm,
	W =180.000 deg,	P =   0.000 deg,	R =    90.000 deg
};
P[9493]{
   GP1:
	UF : 1, UT : 1,		CONFIG : 'N U T, 0, 0, 1',
	X =  85.000  mm,	Y =  205.000  mm,	Z =   15.000 mm,
	W =180.000 deg,	P =   0.000 deg,	R =    90.000 deg
};
P[9494]{
   GP1:
	UF : 1, UT : 1,		CONFIG : 'N U T, 0, 0, 1',
	X =  85.000  mm,	Y =  205.000  mm,	Z =   0.600 mm,
	W =180.000 deg,	P =   0.000 deg,	R =    90.000 deg
};
P[9495]{
   GP1:
	UF : 1, UT : 1,		CONFIG : 'N U T, 0, 0, 1',
	X =  85.000  mm,	Y =  205.000  mm,	Z =   15.000 mm,
	W =180.000 deg,	P =   0.000 deg,	R =    90.000 deg
};
P[9496]{
   GP1:
	UF : 1, UT : 1,		CONFIG : 'N U T, 0, 0, 1',
	X =  88.000  mm,	Y =  205.000  mm,	Z =   15.000 mm,
	W =180.000 deg,	P =   0.000 deg,	R =    90.000 deg
};
P[9497]{
   GP1:
	UF : 1, UT : 1,		CONFIG : 'N U T, 0, 0, 1',
	X =  88.000  mm,	Y =  205.000  mm,	Z =   0.600 mm,
	W =180.000 deg,	P =   0.000 deg,	R =    90.000 deg
};
P[9498]{
   GP1:
	UF : 1, UT : 1,		CONFIG : 'N U T, 0, 0, 1',
	X =  88.000  mm,	Y =  205.000  mm,	Z =   15.000 mm,
	W =180.000 deg,	P =   0.000 deg,	R =    90.000 deg
};
P[9499]{
   GP1:
	UF : 1, UT : 1,		CONFIG : 'N U T, 0, 0, 1',
	X =  91.000  mm,	Y =  205.000  mm,	Z =   15.000 mm,
	W =180.000 deg,	P =   0.000 deg,	R =    90.000 deg
};
P[9500]{
   GP1:
	UF : 1, UT : 1,		CONFIG : 'N U T, 0, 0, 1',
	X =  91.000  mm,	Y =  205.000  mm,	Z =   0.600 mm,
	W =180.000 deg,	P =   0.000 deg,	R =    90.000 deg
};
P[9501]{
   GP1:
	UF : 1, UT : 1,		CONFIG : 'N U T, 0, 0, 1',
	X =  91.000  mm,	Y =  205.000  mm,	Z =   15.000 mm,
	W =180.000 deg,	P =   0.000 deg,	R =    90.000 deg
};
P[9502]{
   GP1:
	UF : 1, UT : 1,		CONFIG : 'N U T, 0, 0, 1',
	X =  94.000  mm,	Y =  205.000  mm,	Z =   15.000 mm,
	W =180.000 deg,	P =   0.000 deg,	R =    90.000 deg
};
P[9503]{
   GP1:
	UF : 1, UT : 1,		CONFIG : 'N U T, 0, 0, 1',
	X =  94.000  mm,	Y =  205.000  mm,	Z =   0.600 mm,
	W =180.000 deg,	P =   0.000 deg,	R =    90.000 deg
};
P[9504]{
   GP1:
	UF : 1, UT : 1,		CONFIG : 'N U T, 0, 0, 1',
	X =  94.000  mm,	Y =  205.000  mm,	Z =   15.000 mm,
	W =180.000 deg,	P =   0.000 deg,	R =    90.000 deg
};
P[9505]{
   GP1:
	UF : 1, UT : 1,		CONFIG : 'N U T, 0, 0, 1',
	X =  97.000  mm,	Y =  205.000  mm,	Z =   15.000 mm,
	W =180.000 deg,	P =   0.000 deg,	R =    90.000 deg
};
P[9506]{
   GP1:
	UF : 1, UT : 1,		CONFIG : 'N U T, 0, 0, 1',
	X =  97.000  mm,	Y =  205.000  mm,	Z =   0.600 mm,
	W =180.000 deg,	P =   0.000 deg,	R =    90.000 deg
};
P[9507]{
   GP1:
	UF : 1, UT : 1,		CONFIG : 'N U T, 0, 0, 1',
	X =  97.000  mm,	Y =  205.000  mm,	Z =   15.000 mm,
	W =180.000 deg,	P =   0.000 deg,	R =    90.000 deg
};
P[9508]{
   GP1:
	UF : 1, UT : 1,		CONFIG : 'N U T, 0, 0, 1',
	X =  100.000  mm,	Y =  205.000  mm,	Z =   15.000 mm,
	W =180.000 deg,	P =   0.000 deg,	R =    90.000 deg
};
P[9509]{
   GP1:
	UF : 1, UT : 1,		CONFIG : 'N U T, 0, 0, 1',
	X =  100.000  mm,	Y =  205.000  mm,	Z =   0.600 mm,
	W =180.000 deg,	P =   0.000 deg,	R =    90.000 deg
};
P[9510]{
   GP1:
	UF : 1, UT : 1,		CONFIG : 'N U T, 0, 0, 1',
	X =  100.000  mm,	Y =  205.000  mm,	Z =   15.000 mm,
	W =180.000 deg,	P =   0.000 deg,	R =    90.000 deg
};
P[9511]{
   GP1:
	UF : 1, UT : 1,		CONFIG : 'N U T, 0, 0, 1',
	X =  103.000  mm,	Y =  205.000  mm,	Z =   15.000 mm,
	W =180.000 deg,	P =   0.000 deg,	R =    90.000 deg
};
P[9512]{
   GP1:
	UF : 1, UT : 1,		CONFIG : 'N U T, 0, 0, 1',
	X =  103.000  mm,	Y =  205.000  mm,	Z =   0.600 mm,
	W =180.000 deg,	P =   0.000 deg,	R =    90.000 deg
};
P[9513]{
   GP1:
	UF : 1, UT : 1,		CONFIG : 'N U T, 0, 0, 1',
	X =  103.000  mm,	Y =  205.000  mm,	Z =   15.000 mm,
	W =180.000 deg,	P =   0.000 deg,	R =    90.000 deg
};
P[9514]{
   GP1:
	UF : 1, UT : 1,		CONFIG : 'N U T, 0, 0, 1',
	X =  106.000  mm,	Y =  205.000  mm,	Z =   15.000 mm,
	W =180.000 deg,	P =   0.000 deg,	R =    90.000 deg
};
P[9515]{
   GP1:
	UF : 1, UT : 1,		CONFIG : 'N U T, 0, 0, 1',
	X =  106.000  mm,	Y =  205.000  mm,	Z =   0.600 mm,
	W =180.000 deg,	P =   0.000 deg,	R =    90.000 deg
};
P[9516]{
   GP1:
	UF : 1, UT : 1,		CONFIG : 'N U T, 0, 0, 1',
	X =  106.000  mm,	Y =  205.000  mm,	Z =   15.000 mm,
	W =180.000 deg,	P =   0.000 deg,	R =    90.000 deg
};
P[9517]{
   GP1:
	UF : 1, UT : 1,		CONFIG : 'N U T, 0, 0, 1',
	X =  109.000  mm,	Y =  205.000  mm,	Z =   15.000 mm,
	W =180.000 deg,	P =   0.000 deg,	R =    90.000 deg
};
P[9518]{
   GP1:
	UF : 1, UT : 1,		CONFIG : 'N U T, 0, 0, 1',
	X =  109.000  mm,	Y =  205.000  mm,	Z =   0.600 mm,
	W =180.000 deg,	P =   0.000 deg,	R =    90.000 deg
};
P[9519]{
   GP1:
	UF : 1, UT : 1,		CONFIG : 'N U T, 0, 0, 1',
	X =  109.000  mm,	Y =  205.000  mm,	Z =   15.000 mm,
	W =180.000 deg,	P =   0.000 deg,	R =    90.000 deg
};
P[9520]{
   GP1:
	UF : 1, UT : 1,		CONFIG : 'N U T, 0, 0, 1',
	X =  112.000  mm,	Y =  205.000  mm,	Z =   15.000 mm,
	W =180.000 deg,	P =   0.000 deg,	R =    90.000 deg
};
P[9521]{
   GP1:
	UF : 1, UT : 1,		CONFIG : 'N U T, 0, 0, 1',
	X =  112.000  mm,	Y =  205.000  mm,	Z =   0.600 mm,
	W =180.000 deg,	P =   0.000 deg,	R =    90.000 deg
};
P[9522]{
   GP1:
	UF : 1, UT : 1,		CONFIG : 'N U T, 0, 0, 1',
	X =  112.000  mm,	Y =  205.000  mm,	Z =   15.000 mm,
	W =180.000 deg,	P =   0.000 deg,	R =    90.000 deg
};
P[9523]{
   GP1:
	UF : 1, UT : 1,		CONFIG : 'N U T, 0, 0, 1',
	X =  115.000  mm,	Y =  205.000  mm,	Z =   15.000 mm,
	W =180.000 deg,	P =   0.000 deg,	R =    90.000 deg
};
P[9524]{
   GP1:
	UF : 1, UT : 1,		CONFIG : 'N U T, 0, 0, 1',
	X =  115.000  mm,	Y =  205.000  mm,	Z =   0.600 mm,
	W =180.000 deg,	P =   0.000 deg,	R =    90.000 deg
};
P[9525]{
   GP1:
	UF : 1, UT : 1,		CONFIG : 'N U T, 0, 0, 1',
	X =  115.000  mm,	Y =  205.000  mm,	Z =   15.000 mm,
	W =180.000 deg,	P =   0.000 deg,	R =    90.000 deg
};
P[9526]{
   GP1:
	UF : 1, UT : 1,		CONFIG : 'N U T, 0, 0, 1',
	X =  118.000  mm,	Y =  205.000  mm,	Z =   15.000 mm,
	W =180.000 deg,	P =   0.000 deg,	R =    90.000 deg
};
P[9527]{
   GP1:
	UF : 1, UT : 1,		CONFIG : 'N U T, 0, 0, 1',
	X =  118.000  mm,	Y =  205.000  mm,	Z =   0.600 mm,
	W =180.000 deg,	P =   0.000 deg,	R =    90.000 deg
};
P[9528]{
   GP1:
	UF : 1, UT : 1,		CONFIG : 'N U T, 0, 0, 1',
	X =  118.000  mm,	Y =  205.000  mm,	Z =   15.000 mm,
	W =180.000 deg,	P =   0.000 deg,	R =    90.000 deg
};
P[9529]{
   GP1:
	UF : 1, UT : 1,		CONFIG : 'N U T, 0, 0, 1',
	X =  121.000  mm,	Y =  205.000  mm,	Z =   15.000 mm,
	W =180.000 deg,	P =   0.000 deg,	R =    90.000 deg
};
P[9530]{
   GP1:
	UF : 1, UT : 1,		CONFIG : 'N U T, 0, 0, 1',
	X =  121.000  mm,	Y =  205.000  mm,	Z =   0.600 mm,
	W =180.000 deg,	P =   0.000 deg,	R =    90.000 deg
};
P[9531]{
   GP1:
	UF : 1, UT : 1,		CONFIG : 'N U T, 0, 0, 1',
	X =  121.000  mm,	Y =  205.000  mm,	Z =   15.000 mm,
	W =180.000 deg,	P =   0.000 deg,	R =    90.000 deg
};
P[9532]{
   GP1:
	UF : 1, UT : 1,		CONFIG : 'N U T, 0, 0, 1',
	X =  124.000  mm,	Y =  205.000  mm,	Z =   15.000 mm,
	W =180.000 deg,	P =   0.000 deg,	R =    90.000 deg
};
P[9533]{
   GP1:
	UF : 1, UT : 1,		CONFIG : 'N U T, 0, 0, 1',
	X =  124.000  mm,	Y =  205.000  mm,	Z =   0.600 mm,
	W =180.000 deg,	P =   0.000 deg,	R =    90.000 deg
};
P[9534]{
   GP1:
	UF : 1, UT : 1,		CONFIG : 'N U T, 0, 0, 1',
	X =  124.000  mm,	Y =  205.000  mm,	Z =   15.000 mm,
	W =180.000 deg,	P =   0.000 deg,	R =    90.000 deg
};
P[9535]{
   GP1:
	UF : 1, UT : 1,		CONFIG : 'N U T, 0, 0, 1',
	X =  127.000  mm,	Y =  205.000  mm,	Z =   15.000 mm,
	W =180.000 deg,	P =   0.000 deg,	R =    90.000 deg
};
P[9536]{
   GP1:
	UF : 1, UT : 1,		CONFIG : 'N U T, 0, 0, 1',
	X =  127.000  mm,	Y =  205.000  mm,	Z =   0.600 mm,
	W =180.000 deg,	P =   0.000 deg,	R =    90.000 deg
};
P[9537]{
   GP1:
	UF : 1, UT : 1,		CONFIG : 'N U T, 0, 0, 1',
	X =  127.000  mm,	Y =  205.000  mm,	Z =   15.000 mm,
	W =180.000 deg,	P =   0.000 deg,	R =    90.000 deg
};
P[9538]{
   GP1:
	UF : 1, UT : 1,		CONFIG : 'N U T, 0, 0, 1',
	X =  130.000  mm,	Y =  205.000  mm,	Z =   15.000 mm,
	W =180.000 deg,	P =   0.000 deg,	R =    90.000 deg
};
P[9539]{
   GP1:
	UF : 1, UT : 1,		CONFIG : 'N U T, 0, 0, 1',
	X =  130.000  mm,	Y =  205.000  mm,	Z =   0.600 mm,
	W =180.000 deg,	P =   0.000 deg,	R =    90.000 deg
};
P[9540]{
   GP1:
	UF : 1, UT : 1,		CONFIG : 'N U T, 0, 0, 1',
	X =  130.000  mm,	Y =  205.000  mm,	Z =   15.000 mm,
	W =180.000 deg,	P =   0.000 deg,	R =    90.000 deg
};
P[9541]{
   GP1:
	UF : 1, UT : 1,		CONFIG : 'N U T, 0, 0, 1',
	X =  133.000  mm,	Y =  205.000  mm,	Z =   15.000 mm,
	W =180.000 deg,	P =   0.000 deg,	R =    90.000 deg
};
P[9542]{
   GP1:
	UF : 1, UT : 1,		CONFIG : 'N U T, 0, 0, 1',
	X =  133.000  mm,	Y =  205.000  mm,	Z =   0.600 mm,
	W =180.000 deg,	P =   0.000 deg,	R =    90.000 deg
};
P[9543]{
   GP1:
	UF : 1, UT : 1,		CONFIG : 'N U T, 0, 0, 1',
	X =  133.000  mm,	Y =  205.000  mm,	Z =   15.000 mm,
	W =180.000 deg,	P =   0.000 deg,	R =    90.000 deg
};
P[9544]{
   GP1:
	UF : 1, UT : 1,		CONFIG : 'N U T, 0, 0, 1',
	X =  136.000  mm,	Y =  205.000  mm,	Z =   15.000 mm,
	W =180.000 deg,	P =   0.000 deg,	R =    90.000 deg
};
P[9545]{
   GP1:
	UF : 1, UT : 1,		CONFIG : 'N U T, 0, 0, 1',
	X =  136.000  mm,	Y =  205.000  mm,	Z =   0.600 mm,
	W =180.000 deg,	P =   0.000 deg,	R =    90.000 deg
};
P[9546]{
   GP1:
	UF : 1, UT : 1,		CONFIG : 'N U T, 0, 0, 1',
	X =  136.000  mm,	Y =  205.000  mm,	Z =   15.000 mm,
	W =180.000 deg,	P =   0.000 deg,	R =    90.000 deg
};
P[9547]{
   GP1:
	UF : 1, UT : 1,		CONFIG : 'N U T, 0, 0, 1',
	X =  139.000  mm,	Y =  205.000  mm,	Z =   15.000 mm,
	W =180.000 deg,	P =   0.000 deg,	R =    90.000 deg
};
P[9548]{
   GP1:
	UF : 1, UT : 1,		CONFIG : 'N U T, 0, 0, 1',
	X =  139.000  mm,	Y =  205.000  mm,	Z =   0.600 mm,
	W =180.000 deg,	P =   0.000 deg,	R =    90.000 deg
};
P[9549]{
   GP1:
	UF : 1, UT : 1,		CONFIG : 'N U T, 0, 0, 1',
	X =  139.000  mm,	Y =  205.000  mm,	Z =   15.000 mm,
	W =180.000 deg,	P =   0.000 deg,	R =    90.000 deg
};
P[9550]{
   GP1:
	UF : 1, UT : 1,		CONFIG : 'N U T, 0, 0, 1',
	X =  142.000  mm,	Y =  205.000  mm,	Z =   15.000 mm,
	W =180.000 deg,	P =   0.000 deg,	R =    90.000 deg
};
P[9551]{
   GP1:
	UF : 1, UT : 1,		CONFIG : 'N U T, 0, 0, 1',
	X =  142.000  mm,	Y =  205.000  mm,	Z =   0.600 mm,
	W =180.000 deg,	P =   0.000 deg,	R =    90.000 deg
};
P[9552]{
   GP1:
	UF : 1, UT : 1,		CONFIG : 'N U T, 0, 0, 1',
	X =  142.000  mm,	Y =  205.000  mm,	Z =   15.000 mm,
	W =180.000 deg,	P =   0.000 deg,	R =    90.000 deg
};
P[9553]{
   GP1:
	UF : 1, UT : 1,		CONFIG : 'N U T, 0, 0, 1',
	X =  145.000  mm,	Y =  205.000  mm,	Z =   15.000 mm,
	W =180.000 deg,	P =   0.000 deg,	R =    90.000 deg
};
P[9554]{
   GP1:
	UF : 1, UT : 1,		CONFIG : 'N U T, 0, 0, 1',
	X =  145.000  mm,	Y =  205.000  mm,	Z =   0.600 mm,
	W =180.000 deg,	P =   0.000 deg,	R =    90.000 deg
};
P[9555]{
   GP1:
	UF : 1, UT : 1,		CONFIG : 'N U T, 0, 0, 1',
	X =  145.000  mm,	Y =  205.000  mm,	Z =   15.000 mm,
	W =180.000 deg,	P =   0.000 deg,	R =    90.000 deg
};
P[9556]{
   GP1:
	UF : 1, UT : 1,		CONFIG : 'N U T, 0, 0, 1',
	X =  148.000  mm,	Y =  205.000  mm,	Z =   15.000 mm,
	W =180.000 deg,	P =   0.000 deg,	R =    90.000 deg
};
P[9557]{
   GP1:
	UF : 1, UT : 1,		CONFIG : 'N U T, 0, 0, 1',
	X =  148.000  mm,	Y =  205.000  mm,	Z =   0.600 mm,
	W =180.000 deg,	P =   0.000 deg,	R =    90.000 deg
};
P[9558]{
   GP1:
	UF : 1, UT : 1,		CONFIG : 'N U T, 0, 0, 1',
	X =  148.000  mm,	Y =  205.000  mm,	Z =   15.000 mm,
	W =180.000 deg,	P =   0.000 deg,	R =    90.000 deg
};
P[9559]{
   GP1:
	UF : 1, UT : 1,		CONFIG : 'N U T, 0, 0, 1',
	X =  151.000  mm,	Y =  205.000  mm,	Z =   15.000 mm,
	W =180.000 deg,	P =   0.000 deg,	R =    90.000 deg
};
P[9560]{
   GP1:
	UF : 1, UT : 1,		CONFIG : 'N U T, 0, 0, 1',
	X =  151.000  mm,	Y =  205.000  mm,	Z =   0.600 mm,
	W =180.000 deg,	P =   0.000 deg,	R =    90.000 deg
};
P[9561]{
   GP1:
	UF : 1, UT : 1,		CONFIG : 'N U T, 0, 0, 1',
	X =  151.000  mm,	Y =  205.000  mm,	Z =   15.000 mm,
	W =180.000 deg,	P =   0.000 deg,	R =    90.000 deg
};
P[9562]{
   GP1:
	UF : 1, UT : 1,		CONFIG : 'N U T, 0, 0, 1',
	X =  154.000  mm,	Y =  205.000  mm,	Z =   15.000 mm,
	W =180.000 deg,	P =   0.000 deg,	R =    90.000 deg
};
P[9563]{
   GP1:
	UF : 1, UT : 1,		CONFIG : 'N U T, 0, 0, 1',
	X =  154.000  mm,	Y =  205.000  mm,	Z =   0.600 mm,
	W =180.000 deg,	P =   0.000 deg,	R =    90.000 deg
};
P[9564]{
   GP1:
	UF : 1, UT : 1,		CONFIG : 'N U T, 0, 0, 1',
	X =  154.000  mm,	Y =  205.000  mm,	Z =   15.000 mm,
	W =180.000 deg,	P =   0.000 deg,	R =    90.000 deg
};
P[9565]{
   GP1:
	UF : 1, UT : 1,		CONFIG : 'N U T, 0, 0, 1',
	X =  157.000  mm,	Y =  205.000  mm,	Z =   15.000 mm,
	W =180.000 deg,	P =   0.000 deg,	R =    90.000 deg
};
P[9566]{
   GP1:
	UF : 1, UT : 1,		CONFIG : 'N U T, 0, 0, 1',
	X =  157.000  mm,	Y =  205.000  mm,	Z =   0.600 mm,
	W =180.000 deg,	P =   0.000 deg,	R =    90.000 deg
};
P[9567]{
   GP1:
	UF : 1, UT : 1,		CONFIG : 'N U T, 0, 0, 1',
	X =  157.000  mm,	Y =  205.000  mm,	Z =   15.000 mm,
	W =180.000 deg,	P =   0.000 deg,	R =    90.000 deg
};
P[9568]{
   GP1:
	UF : 1, UT : 1,		CONFIG : 'N U T, 0, 0, 1',
	X =  160.000  mm,	Y =  205.000  mm,	Z =   15.000 mm,
	W =180.000 deg,	P =   0.000 deg,	R =    90.000 deg
};
P[9569]{
   GP1:
	UF : 1, UT : 1,		CONFIG : 'N U T, 0, 0, 1',
	X =  160.000  mm,	Y =  205.000  mm,	Z =   0.600 mm,
	W =180.000 deg,	P =   0.000 deg,	R =    90.000 deg
};
P[9570]{
   GP1:
	UF : 1, UT : 1,		CONFIG : 'N U T, 0, 0, 1',
	X =  160.000  mm,	Y =  205.000  mm,	Z =   15.000 mm,
	W =180.000 deg,	P =   0.000 deg,	R =    90.000 deg
};
P[9571]{
   GP1:
	UF : 1, UT : 1,		CONFIG : 'N U T, 0, 0, 1',
	X =  163.000  mm,	Y =  205.000  mm,	Z =   15.000 mm,
	W =180.000 deg,	P =   0.000 deg,	R =    90.000 deg
};
P[9572]{
   GP1:
	UF : 1, UT : 1,		CONFIG : 'N U T, 0, 0, 1',
	X =  163.000  mm,	Y =  205.000  mm,	Z =   0.600 mm,
	W =180.000 deg,	P =   0.000 deg,	R =    90.000 deg
};
P[9573]{
   GP1:
	UF : 1, UT : 1,		CONFIG : 'N U T, 0, 0, 1',
	X =  163.000  mm,	Y =  205.000  mm,	Z =   15.000 mm,
	W =180.000 deg,	P =   0.000 deg,	R =    90.000 deg
};
P[9574]{
   GP1:
	UF : 1, UT : 1,		CONFIG : 'N U T, 0, 0, 1',
	X =  166.000  mm,	Y =  205.000  mm,	Z =   15.000 mm,
	W =180.000 deg,	P =   0.000 deg,	R =    90.000 deg
};
P[9575]{
   GP1:
	UF : 1, UT : 1,		CONFIG : 'N U T, 0, 0, 1',
	X =  166.000  mm,	Y =  205.000  mm,	Z =   0.600 mm,
	W =180.000 deg,	P =   0.000 deg,	R =    90.000 deg
};
P[9576]{
   GP1:
	UF : 1, UT : 1,		CONFIG : 'N U T, 0, 0, 1',
	X =  166.000  mm,	Y =  205.000  mm,	Z =   15.000 mm,
	W =180.000 deg,	P =   0.000 deg,	R =    90.000 deg
};
P[9577]{
   GP1:
	UF : 1, UT : 1,		CONFIG : 'N U T, 0, 0, 1',
	X =  169.000  mm,	Y =  205.000  mm,	Z =   15.000 mm,
	W =180.000 deg,	P =   0.000 deg,	R =    90.000 deg
};
P[9578]{
   GP1:
	UF : 1, UT : 1,		CONFIG : 'N U T, 0, 0, 1',
	X =  169.000  mm,	Y =  205.000  mm,	Z =   0.600 mm,
	W =180.000 deg,	P =   0.000 deg,	R =    90.000 deg
};
P[9579]{
   GP1:
	UF : 1, UT : 1,		CONFIG : 'N U T, 0, 0, 1',
	X =  169.000  mm,	Y =  205.000  mm,	Z =   15.000 mm,
	W =180.000 deg,	P =   0.000 deg,	R =    90.000 deg
};
P[9580]{
   GP1:
	UF : 1, UT : 1,		CONFIG : 'N U T, 0, 0, 1',
	X =  172.000  mm,	Y =  205.000  mm,	Z =   15.000 mm,
	W =180.000 deg,	P =   0.000 deg,	R =    90.000 deg
};
P[9581]{
   GP1:
	UF : 1, UT : 1,		CONFIG : 'N U T, 0, 0, 1',
	X =  172.000  mm,	Y =  205.000  mm,	Z =   0.600 mm,
	W =180.000 deg,	P =   0.000 deg,	R =    90.000 deg
};
P[9582]{
   GP1:
	UF : 1, UT : 1,		CONFIG : 'N U T, 0, 0, 1',
	X =  172.000  mm,	Y =  205.000  mm,	Z =   15.000 mm,
	W =180.000 deg,	P =   0.000 deg,	R =    90.000 deg
};
P[9583]{
   GP1:
	UF : 1, UT : 1,		CONFIG : 'N U T, 0, 0, 1',
	X =  175.000  mm,	Y =  205.000  mm,	Z =   15.000 mm,
	W =180.000 deg,	P =   0.000 deg,	R =    90.000 deg
};
P[9584]{
   GP1:
	UF : 1, UT : 1,		CONFIG : 'N U T, 0, 0, 1',
	X =  175.000  mm,	Y =  205.000  mm,	Z =   0.600 mm,
	W =180.000 deg,	P =   0.000 deg,	R =    90.000 deg
};
P[9585]{
   GP1:
	UF : 1, UT : 1,		CONFIG : 'N U T, 0, 0, 1',
	X =  175.000  mm,	Y =  205.000  mm,	Z =   15.000 mm,
	W =180.000 deg,	P =   0.000 deg,	R =    90.000 deg
};
P[9586]{
   GP1:
	UF : 1, UT : 1,		CONFIG : 'N U T, 0, 0, 1',
	X =  178.000  mm,	Y =  205.000  mm,	Z =   15.000 mm,
	W =180.000 deg,	P =   0.000 deg,	R =    90.000 deg
};
P[9587]{
   GP1:
	UF : 1, UT : 1,		CONFIG : 'N U T, 0, 0, 1',
	X =  178.000  mm,	Y =  205.000  mm,	Z =   0.600 mm,
	W =180.000 deg,	P =   0.000 deg,	R =    90.000 deg
};
P[9588]{
   GP1:
	UF : 1, UT : 1,		CONFIG : 'N U T, 0, 0, 1',
	X =  178.000  mm,	Y =  205.000  mm,	Z =   15.000 mm,
	W =180.000 deg,	P =   0.000 deg,	R =    90.000 deg
};
P[9589]{
   GP1:
	UF : 1, UT : 1,		CONFIG : 'N U T, 0, 0, 1',
	X =  1.000  mm,	Y =  208.000  mm,	Z =   15.000 mm,
	W =180.000 deg,	P =   0.000 deg,	R =    90.000 deg
};
P[9590]{
   GP1:
	UF : 1, UT : 1,		CONFIG : 'N U T, 0, 0, 1',
	X =  1.000  mm,	Y =  208.000  mm,	Z =   0.600 mm,
	W =180.000 deg,	P =   0.000 deg,	R =    90.000 deg
};
P[9591]{
   GP1:
	UF : 1, UT : 1,		CONFIG : 'N U T, 0, 0, 1',
	X =  1.000  mm,	Y =  208.000  mm,	Z =   15.000 mm,
	W =180.000 deg,	P =   0.000 deg,	R =    90.000 deg
};
P[9592]{
   GP1:
	UF : 1, UT : 1,		CONFIG : 'N U T, 0, 0, 1',
	X =  4.000  mm,	Y =  208.000  mm,	Z =   15.000 mm,
	W =180.000 deg,	P =   0.000 deg,	R =    90.000 deg
};
P[9593]{
   GP1:
	UF : 1, UT : 1,		CONFIG : 'N U T, 0, 0, 1',
	X =  4.000  mm,	Y =  208.000  mm,	Z =   0.600 mm,
	W =180.000 deg,	P =   0.000 deg,	R =    90.000 deg
};
P[9594]{
   GP1:
	UF : 1, UT : 1,		CONFIG : 'N U T, 0, 0, 1',
	X =  4.000  mm,	Y =  208.000  mm,	Z =   15.000 mm,
	W =180.000 deg,	P =   0.000 deg,	R =    90.000 deg
};
P[9595]{
   GP1:
	UF : 1, UT : 1,		CONFIG : 'N U T, 0, 0, 1',
	X =  7.000  mm,	Y =  208.000  mm,	Z =   15.000 mm,
	W =180.000 deg,	P =   0.000 deg,	R =    90.000 deg
};
P[9596]{
   GP1:
	UF : 1, UT : 1,		CONFIG : 'N U T, 0, 0, 1',
	X =  7.000  mm,	Y =  208.000  mm,	Z =   0.600 mm,
	W =180.000 deg,	P =   0.000 deg,	R =    90.000 deg
};
P[9597]{
   GP1:
	UF : 1, UT : 1,		CONFIG : 'N U T, 0, 0, 1',
	X =  7.000  mm,	Y =  208.000  mm,	Z =   15.000 mm,
	W =180.000 deg,	P =   0.000 deg,	R =    90.000 deg
};
P[9598]{
   GP1:
	UF : 1, UT : 1,		CONFIG : 'N U T, 0, 0, 1',
	X =  10.000  mm,	Y =  208.000  mm,	Z =   15.000 mm,
	W =180.000 deg,	P =   0.000 deg,	R =    90.000 deg
};
P[9599]{
   GP1:
	UF : 1, UT : 1,		CONFIG : 'N U T, 0, 0, 1',
	X =  10.000  mm,	Y =  208.000  mm,	Z =   0.600 mm,
	W =180.000 deg,	P =   0.000 deg,	R =    90.000 deg
};
P[9600]{
   GP1:
	UF : 1, UT : 1,		CONFIG : 'N U T, 0, 0, 1',
	X =  10.000  mm,	Y =  208.000  mm,	Z =   15.000 mm,
	W =180.000 deg,	P =   0.000 deg,	R =    90.000 deg
};
P[9601]{
   GP1:
	UF : 1, UT : 1,		CONFIG : 'N U T, 0, 0, 1',
	X =  13.000  mm,	Y =  208.000  mm,	Z =   15.000 mm,
	W =180.000 deg,	P =   0.000 deg,	R =    90.000 deg
};
P[9602]{
   GP1:
	UF : 1, UT : 1,		CONFIG : 'N U T, 0, 0, 1',
	X =  13.000  mm,	Y =  208.000  mm,	Z =   0.600 mm,
	W =180.000 deg,	P =   0.000 deg,	R =    90.000 deg
};
P[9603]{
   GP1:
	UF : 1, UT : 1,		CONFIG : 'N U T, 0, 0, 1',
	X =  13.000  mm,	Y =  208.000  mm,	Z =   15.000 mm,
	W =180.000 deg,	P =   0.000 deg,	R =    90.000 deg
};
P[9604]{
   GP1:
	UF : 1, UT : 1,		CONFIG : 'N U T, 0, 0, 1',
	X =  16.000  mm,	Y =  208.000  mm,	Z =   15.000 mm,
	W =180.000 deg,	P =   0.000 deg,	R =    90.000 deg
};
P[9605]{
   GP1:
	UF : 1, UT : 1,		CONFIG : 'N U T, 0, 0, 1',
	X =  16.000  mm,	Y =  208.000  mm,	Z =   0.600 mm,
	W =180.000 deg,	P =   0.000 deg,	R =    90.000 deg
};
P[9606]{
   GP1:
	UF : 1, UT : 1,		CONFIG : 'N U T, 0, 0, 1',
	X =  16.000  mm,	Y =  208.000  mm,	Z =   15.000 mm,
	W =180.000 deg,	P =   0.000 deg,	R =    90.000 deg
};
P[9607]{
   GP1:
	UF : 1, UT : 1,		CONFIG : 'N U T, 0, 0, 1',
	X =  19.000  mm,	Y =  208.000  mm,	Z =   15.000 mm,
	W =180.000 deg,	P =   0.000 deg,	R =    90.000 deg
};
P[9608]{
   GP1:
	UF : 1, UT : 1,		CONFIG : 'N U T, 0, 0, 1',
	X =  19.000  mm,	Y =  208.000  mm,	Z =   0.600 mm,
	W =180.000 deg,	P =   0.000 deg,	R =    90.000 deg
};
P[9609]{
   GP1:
	UF : 1, UT : 1,		CONFIG : 'N U T, 0, 0, 1',
	X =  19.000  mm,	Y =  208.000  mm,	Z =   15.000 mm,
	W =180.000 deg,	P =   0.000 deg,	R =    90.000 deg
};
P[9610]{
   GP1:
	UF : 1, UT : 1,		CONFIG : 'N U T, 0, 0, 1',
	X =  22.000  mm,	Y =  208.000  mm,	Z =   15.000 mm,
	W =180.000 deg,	P =   0.000 deg,	R =    90.000 deg
};
P[9611]{
   GP1:
	UF : 1, UT : 1,		CONFIG : 'N U T, 0, 0, 1',
	X =  22.000  mm,	Y =  208.000  mm,	Z =   0.600 mm,
	W =180.000 deg,	P =   0.000 deg,	R =    90.000 deg
};
P[9612]{
   GP1:
	UF : 1, UT : 1,		CONFIG : 'N U T, 0, 0, 1',
	X =  22.000  mm,	Y =  208.000  mm,	Z =   15.000 mm,
	W =180.000 deg,	P =   0.000 deg,	R =    90.000 deg
};
P[9613]{
   GP1:
	UF : 1, UT : 1,		CONFIG : 'N U T, 0, 0, 1',
	X =  25.000  mm,	Y =  208.000  mm,	Z =   15.000 mm,
	W =180.000 deg,	P =   0.000 deg,	R =    90.000 deg
};
P[9614]{
   GP1:
	UF : 1, UT : 1,		CONFIG : 'N U T, 0, 0, 1',
	X =  25.000  mm,	Y =  208.000  mm,	Z =   0.600 mm,
	W =180.000 deg,	P =   0.000 deg,	R =    90.000 deg
};
P[9615]{
   GP1:
	UF : 1, UT : 1,		CONFIG : 'N U T, 0, 0, 1',
	X =  25.000  mm,	Y =  208.000  mm,	Z =   15.000 mm,
	W =180.000 deg,	P =   0.000 deg,	R =    90.000 deg
};
P[9616]{
   GP1:
	UF : 1, UT : 1,		CONFIG : 'N U T, 0, 0, 1',
	X =  28.000  mm,	Y =  208.000  mm,	Z =   15.000 mm,
	W =180.000 deg,	P =   0.000 deg,	R =    90.000 deg
};
P[9617]{
   GP1:
	UF : 1, UT : 1,		CONFIG : 'N U T, 0, 0, 1',
	X =  28.000  mm,	Y =  208.000  mm,	Z =   0.600 mm,
	W =180.000 deg,	P =   0.000 deg,	R =    90.000 deg
};
P[9618]{
   GP1:
	UF : 1, UT : 1,		CONFIG : 'N U T, 0, 0, 1',
	X =  28.000  mm,	Y =  208.000  mm,	Z =   15.000 mm,
	W =180.000 deg,	P =   0.000 deg,	R =    90.000 deg
};
P[9619]{
   GP1:
	UF : 1, UT : 1,		CONFIG : 'N U T, 0, 0, 1',
	X =  31.000  mm,	Y =  208.000  mm,	Z =   15.000 mm,
	W =180.000 deg,	P =   0.000 deg,	R =    90.000 deg
};
P[9620]{
   GP1:
	UF : 1, UT : 1,		CONFIG : 'N U T, 0, 0, 1',
	X =  31.000  mm,	Y =  208.000  mm,	Z =   0.600 mm,
	W =180.000 deg,	P =   0.000 deg,	R =    90.000 deg
};
P[9621]{
   GP1:
	UF : 1, UT : 1,		CONFIG : 'N U T, 0, 0, 1',
	X =  31.000  mm,	Y =  208.000  mm,	Z =   15.000 mm,
	W =180.000 deg,	P =   0.000 deg,	R =    90.000 deg
};
P[9622]{
   GP1:
	UF : 1, UT : 1,		CONFIG : 'N U T, 0, 0, 1',
	X =  34.000  mm,	Y =  208.000  mm,	Z =   15.000 mm,
	W =180.000 deg,	P =   0.000 deg,	R =    90.000 deg
};
P[9623]{
   GP1:
	UF : 1, UT : 1,		CONFIG : 'N U T, 0, 0, 1',
	X =  34.000  mm,	Y =  208.000  mm,	Z =   0.600 mm,
	W =180.000 deg,	P =   0.000 deg,	R =    90.000 deg
};
P[9624]{
   GP1:
	UF : 1, UT : 1,		CONFIG : 'N U T, 0, 0, 1',
	X =  34.000  mm,	Y =  208.000  mm,	Z =   15.000 mm,
	W =180.000 deg,	P =   0.000 deg,	R =    90.000 deg
};
P[9625]{
   GP1:
	UF : 1, UT : 1,		CONFIG : 'N U T, 0, 0, 1',
	X =  37.000  mm,	Y =  208.000  mm,	Z =   15.000 mm,
	W =180.000 deg,	P =   0.000 deg,	R =    90.000 deg
};
P[9626]{
   GP1:
	UF : 1, UT : 1,		CONFIG : 'N U T, 0, 0, 1',
	X =  37.000  mm,	Y =  208.000  mm,	Z =   0.600 mm,
	W =180.000 deg,	P =   0.000 deg,	R =    90.000 deg
};
P[9627]{
   GP1:
	UF : 1, UT : 1,		CONFIG : 'N U T, 0, 0, 1',
	X =  37.000  mm,	Y =  208.000  mm,	Z =   15.000 mm,
	W =180.000 deg,	P =   0.000 deg,	R =    90.000 deg
};
P[9628]{
   GP1:
	UF : 1, UT : 1,		CONFIG : 'N U T, 0, 0, 1',
	X =  40.000  mm,	Y =  208.000  mm,	Z =   15.000 mm,
	W =180.000 deg,	P =   0.000 deg,	R =    90.000 deg
};
P[9629]{
   GP1:
	UF : 1, UT : 1,		CONFIG : 'N U T, 0, 0, 1',
	X =  40.000  mm,	Y =  208.000  mm,	Z =   0.600 mm,
	W =180.000 deg,	P =   0.000 deg,	R =    90.000 deg
};
P[9630]{
   GP1:
	UF : 1, UT : 1,		CONFIG : 'N U T, 0, 0, 1',
	X =  40.000  mm,	Y =  208.000  mm,	Z =   15.000 mm,
	W =180.000 deg,	P =   0.000 deg,	R =    90.000 deg
};
P[9631]{
   GP1:
	UF : 1, UT : 1,		CONFIG : 'N U T, 0, 0, 1',
	X =  43.000  mm,	Y =  208.000  mm,	Z =   15.000 mm,
	W =180.000 deg,	P =   0.000 deg,	R =    90.000 deg
};
P[9632]{
   GP1:
	UF : 1, UT : 1,		CONFIG : 'N U T, 0, 0, 1',
	X =  43.000  mm,	Y =  208.000  mm,	Z =   0.600 mm,
	W =180.000 deg,	P =   0.000 deg,	R =    90.000 deg
};
P[9633]{
   GP1:
	UF : 1, UT : 1,		CONFIG : 'N U T, 0, 0, 1',
	X =  43.000  mm,	Y =  208.000  mm,	Z =   15.000 mm,
	W =180.000 deg,	P =   0.000 deg,	R =    90.000 deg
};
P[9634]{
   GP1:
	UF : 1, UT : 1,		CONFIG : 'N U T, 0, 0, 1',
	X =  46.000  mm,	Y =  208.000  mm,	Z =   15.000 mm,
	W =180.000 deg,	P =   0.000 deg,	R =    90.000 deg
};
P[9635]{
   GP1:
	UF : 1, UT : 1,		CONFIG : 'N U T, 0, 0, 1',
	X =  46.000  mm,	Y =  208.000  mm,	Z =   0.600 mm,
	W =180.000 deg,	P =   0.000 deg,	R =    90.000 deg
};
P[9636]{
   GP1:
	UF : 1, UT : 1,		CONFIG : 'N U T, 0, 0, 1',
	X =  46.000  mm,	Y =  208.000  mm,	Z =   15.000 mm,
	W =180.000 deg,	P =   0.000 deg,	R =    90.000 deg
};
P[9637]{
   GP1:
	UF : 1, UT : 1,		CONFIG : 'N U T, 0, 0, 1',
	X =  49.000  mm,	Y =  208.000  mm,	Z =   15.000 mm,
	W =180.000 deg,	P =   0.000 deg,	R =    90.000 deg
};
P[9638]{
   GP1:
	UF : 1, UT : 1,		CONFIG : 'N U T, 0, 0, 1',
	X =  49.000  mm,	Y =  208.000  mm,	Z =   0.600 mm,
	W =180.000 deg,	P =   0.000 deg,	R =    90.000 deg
};
P[9639]{
   GP1:
	UF : 1, UT : 1,		CONFIG : 'N U T, 0, 0, 1',
	X =  49.000  mm,	Y =  208.000  mm,	Z =   15.000 mm,
	W =180.000 deg,	P =   0.000 deg,	R =    90.000 deg
};
P[9640]{
   GP1:
	UF : 1, UT : 1,		CONFIG : 'N U T, 0, 0, 1',
	X =  52.000  mm,	Y =  208.000  mm,	Z =   15.000 mm,
	W =180.000 deg,	P =   0.000 deg,	R =    90.000 deg
};
P[9641]{
   GP1:
	UF : 1, UT : 1,		CONFIG : 'N U T, 0, 0, 1',
	X =  52.000  mm,	Y =  208.000  mm,	Z =   0.600 mm,
	W =180.000 deg,	P =   0.000 deg,	R =    90.000 deg
};
P[9642]{
   GP1:
	UF : 1, UT : 1,		CONFIG : 'N U T, 0, 0, 1',
	X =  52.000  mm,	Y =  208.000  mm,	Z =   15.000 mm,
	W =180.000 deg,	P =   0.000 deg,	R =    90.000 deg
};
P[9643]{
   GP1:
	UF : 1, UT : 1,		CONFIG : 'N U T, 0, 0, 1',
	X =  55.000  mm,	Y =  208.000  mm,	Z =   15.000 mm,
	W =180.000 deg,	P =   0.000 deg,	R =    90.000 deg
};
P[9644]{
   GP1:
	UF : 1, UT : 1,		CONFIG : 'N U T, 0, 0, 1',
	X =  55.000  mm,	Y =  208.000  mm,	Z =   0.600 mm,
	W =180.000 deg,	P =   0.000 deg,	R =    90.000 deg
};
P[9645]{
   GP1:
	UF : 1, UT : 1,		CONFIG : 'N U T, 0, 0, 1',
	X =  55.000  mm,	Y =  208.000  mm,	Z =   15.000 mm,
	W =180.000 deg,	P =   0.000 deg,	R =    90.000 deg
};
P[9646]{
   GP1:
	UF : 1, UT : 1,		CONFIG : 'N U T, 0, 0, 1',
	X =  58.000  mm,	Y =  208.000  mm,	Z =   15.000 mm,
	W =180.000 deg,	P =   0.000 deg,	R =    90.000 deg
};
P[9647]{
   GP1:
	UF : 1, UT : 1,		CONFIG : 'N U T, 0, 0, 1',
	X =  58.000  mm,	Y =  208.000  mm,	Z =   0.600 mm,
	W =180.000 deg,	P =   0.000 deg,	R =    90.000 deg
};
P[9648]{
   GP1:
	UF : 1, UT : 1,		CONFIG : 'N U T, 0, 0, 1',
	X =  58.000  mm,	Y =  208.000  mm,	Z =   15.000 mm,
	W =180.000 deg,	P =   0.000 deg,	R =    90.000 deg
};
P[9649]{
   GP1:
	UF : 1, UT : 1,		CONFIG : 'N U T, 0, 0, 1',
	X =  61.000  mm,	Y =  208.000  mm,	Z =   15.000 mm,
	W =180.000 deg,	P =   0.000 deg,	R =    90.000 deg
};
P[9650]{
   GP1:
	UF : 1, UT : 1,		CONFIG : 'N U T, 0, 0, 1',
	X =  61.000  mm,	Y =  208.000  mm,	Z =   0.600 mm,
	W =180.000 deg,	P =   0.000 deg,	R =    90.000 deg
};
P[9651]{
   GP1:
	UF : 1, UT : 1,		CONFIG : 'N U T, 0, 0, 1',
	X =  61.000  mm,	Y =  208.000  mm,	Z =   15.000 mm,
	W =180.000 deg,	P =   0.000 deg,	R =    90.000 deg
};
P[9652]{
   GP1:
	UF : 1, UT : 1,		CONFIG : 'N U T, 0, 0, 1',
	X =  64.000  mm,	Y =  208.000  mm,	Z =   15.000 mm,
	W =180.000 deg,	P =   0.000 deg,	R =    90.000 deg
};
P[9653]{
   GP1:
	UF : 1, UT : 1,		CONFIG : 'N U T, 0, 0, 1',
	X =  64.000  mm,	Y =  208.000  mm,	Z =   0.600 mm,
	W =180.000 deg,	P =   0.000 deg,	R =    90.000 deg
};
P[9654]{
   GP1:
	UF : 1, UT : 1,		CONFIG : 'N U T, 0, 0, 1',
	X =  64.000  mm,	Y =  208.000  mm,	Z =   15.000 mm,
	W =180.000 deg,	P =   0.000 deg,	R =    90.000 deg
};
P[9655]{
   GP1:
	UF : 1, UT : 1,		CONFIG : 'N U T, 0, 0, 1',
	X =  67.000  mm,	Y =  208.000  mm,	Z =   15.000 mm,
	W =180.000 deg,	P =   0.000 deg,	R =    90.000 deg
};
P[9656]{
   GP1:
	UF : 1, UT : 1,		CONFIG : 'N U T, 0, 0, 1',
	X =  67.000  mm,	Y =  208.000  mm,	Z =   0.600 mm,
	W =180.000 deg,	P =   0.000 deg,	R =    90.000 deg
};
P[9657]{
   GP1:
	UF : 1, UT : 1,		CONFIG : 'N U T, 0, 0, 1',
	X =  67.000  mm,	Y =  208.000  mm,	Z =   15.000 mm,
	W =180.000 deg,	P =   0.000 deg,	R =    90.000 deg
};
P[9658]{
   GP1:
	UF : 1, UT : 1,		CONFIG : 'N U T, 0, 0, 1',
	X =  70.000  mm,	Y =  208.000  mm,	Z =   15.000 mm,
	W =180.000 deg,	P =   0.000 deg,	R =    90.000 deg
};
P[9659]{
   GP1:
	UF : 1, UT : 1,		CONFIG : 'N U T, 0, 0, 1',
	X =  70.000  mm,	Y =  208.000  mm,	Z =   0.600 mm,
	W =180.000 deg,	P =   0.000 deg,	R =    90.000 deg
};
P[9660]{
   GP1:
	UF : 1, UT : 1,		CONFIG : 'N U T, 0, 0, 1',
	X =  70.000  mm,	Y =  208.000  mm,	Z =   15.000 mm,
	W =180.000 deg,	P =   0.000 deg,	R =    90.000 deg
};
P[9661]{
   GP1:
	UF : 1, UT : 1,		CONFIG : 'N U T, 0, 0, 1',
	X =  73.000  mm,	Y =  208.000  mm,	Z =   15.000 mm,
	W =180.000 deg,	P =   0.000 deg,	R =    90.000 deg
};
P[9662]{
   GP1:
	UF : 1, UT : 1,		CONFIG : 'N U T, 0, 0, 1',
	X =  73.000  mm,	Y =  208.000  mm,	Z =   0.600 mm,
	W =180.000 deg,	P =   0.000 deg,	R =    90.000 deg
};
P[9663]{
   GP1:
	UF : 1, UT : 1,		CONFIG : 'N U T, 0, 0, 1',
	X =  73.000  mm,	Y =  208.000  mm,	Z =   15.000 mm,
	W =180.000 deg,	P =   0.000 deg,	R =    90.000 deg
};
P[9664]{
   GP1:
	UF : 1, UT : 1,		CONFIG : 'N U T, 0, 0, 1',
	X =  76.000  mm,	Y =  208.000  mm,	Z =   15.000 mm,
	W =180.000 deg,	P =   0.000 deg,	R =    90.000 deg
};
P[9665]{
   GP1:
	UF : 1, UT : 1,		CONFIG : 'N U T, 0, 0, 1',
	X =  76.000  mm,	Y =  208.000  mm,	Z =   0.600 mm,
	W =180.000 deg,	P =   0.000 deg,	R =    90.000 deg
};
P[9666]{
   GP1:
	UF : 1, UT : 1,		CONFIG : 'N U T, 0, 0, 1',
	X =  76.000  mm,	Y =  208.000  mm,	Z =   15.000 mm,
	W =180.000 deg,	P =   0.000 deg,	R =    90.000 deg
};
P[9667]{
   GP1:
	UF : 1, UT : 1,		CONFIG : 'N U T, 0, 0, 1',
	X =  79.000  mm,	Y =  208.000  mm,	Z =   15.000 mm,
	W =180.000 deg,	P =   0.000 deg,	R =    90.000 deg
};
P[9668]{
   GP1:
	UF : 1, UT : 1,		CONFIG : 'N U T, 0, 0, 1',
	X =  79.000  mm,	Y =  208.000  mm,	Z =   0.600 mm,
	W =180.000 deg,	P =   0.000 deg,	R =    90.000 deg
};
P[9669]{
   GP1:
	UF : 1, UT : 1,		CONFIG : 'N U T, 0, 0, 1',
	X =  79.000  mm,	Y =  208.000  mm,	Z =   15.000 mm,
	W =180.000 deg,	P =   0.000 deg,	R =    90.000 deg
};
P[9670]{
   GP1:
	UF : 1, UT : 1,		CONFIG : 'N U T, 0, 0, 1',
	X =  82.000  mm,	Y =  208.000  mm,	Z =   15.000 mm,
	W =180.000 deg,	P =   0.000 deg,	R =    90.000 deg
};
P[9671]{
   GP1:
	UF : 1, UT : 1,		CONFIG : 'N U T, 0, 0, 1',
	X =  82.000  mm,	Y =  208.000  mm,	Z =   0.600 mm,
	W =180.000 deg,	P =   0.000 deg,	R =    90.000 deg
};
P[9672]{
   GP1:
	UF : 1, UT : 1,		CONFIG : 'N U T, 0, 0, 1',
	X =  82.000  mm,	Y =  208.000  mm,	Z =   15.000 mm,
	W =180.000 deg,	P =   0.000 deg,	R =    90.000 deg
};
P[9673]{
   GP1:
	UF : 1, UT : 1,		CONFIG : 'N U T, 0, 0, 1',
	X =  85.000  mm,	Y =  208.000  mm,	Z =   15.000 mm,
	W =180.000 deg,	P =   0.000 deg,	R =    90.000 deg
};
P[9674]{
   GP1:
	UF : 1, UT : 1,		CONFIG : 'N U T, 0, 0, 1',
	X =  85.000  mm,	Y =  208.000  mm,	Z =   0.600 mm,
	W =180.000 deg,	P =   0.000 deg,	R =    90.000 deg
};
P[9675]{
   GP1:
	UF : 1, UT : 1,		CONFIG : 'N U T, 0, 0, 1',
	X =  85.000  mm,	Y =  208.000  mm,	Z =   15.000 mm,
	W =180.000 deg,	P =   0.000 deg,	R =    90.000 deg
};
P[9676]{
   GP1:
	UF : 1, UT : 1,		CONFIG : 'N U T, 0, 0, 1',
	X =  88.000  mm,	Y =  208.000  mm,	Z =   15.000 mm,
	W =180.000 deg,	P =   0.000 deg,	R =    90.000 deg
};
P[9677]{
   GP1:
	UF : 1, UT : 1,		CONFIG : 'N U T, 0, 0, 1',
	X =  88.000  mm,	Y =  208.000  mm,	Z =   0.600 mm,
	W =180.000 deg,	P =   0.000 deg,	R =    90.000 deg
};
P[9678]{
   GP1:
	UF : 1, UT : 1,		CONFIG : 'N U T, 0, 0, 1',
	X =  88.000  mm,	Y =  208.000  mm,	Z =   15.000 mm,
	W =180.000 deg,	P =   0.000 deg,	R =    90.000 deg
};
P[9679]{
   GP1:
	UF : 1, UT : 1,		CONFIG : 'N U T, 0, 0, 1',
	X =  91.000  mm,	Y =  208.000  mm,	Z =   15.000 mm,
	W =180.000 deg,	P =   0.000 deg,	R =    90.000 deg
};
P[9680]{
   GP1:
	UF : 1, UT : 1,		CONFIG : 'N U T, 0, 0, 1',
	X =  91.000  mm,	Y =  208.000  mm,	Z =   0.600 mm,
	W =180.000 deg,	P =   0.000 deg,	R =    90.000 deg
};
P[9681]{
   GP1:
	UF : 1, UT : 1,		CONFIG : 'N U T, 0, 0, 1',
	X =  91.000  mm,	Y =  208.000  mm,	Z =   15.000 mm,
	W =180.000 deg,	P =   0.000 deg,	R =    90.000 deg
};
P[9682]{
   GP1:
	UF : 1, UT : 1,		CONFIG : 'N U T, 0, 0, 1',
	X =  94.000  mm,	Y =  208.000  mm,	Z =   15.000 mm,
	W =180.000 deg,	P =   0.000 deg,	R =    90.000 deg
};
P[9683]{
   GP1:
	UF : 1, UT : 1,		CONFIG : 'N U T, 0, 0, 1',
	X =  94.000  mm,	Y =  208.000  mm,	Z =   0.600 mm,
	W =180.000 deg,	P =   0.000 deg,	R =    90.000 deg
};
P[9684]{
   GP1:
	UF : 1, UT : 1,		CONFIG : 'N U T, 0, 0, 1',
	X =  94.000  mm,	Y =  208.000  mm,	Z =   15.000 mm,
	W =180.000 deg,	P =   0.000 deg,	R =    90.000 deg
};
P[9685]{
   GP1:
	UF : 1, UT : 1,		CONFIG : 'N U T, 0, 0, 1',
	X =  97.000  mm,	Y =  208.000  mm,	Z =   15.000 mm,
	W =180.000 deg,	P =   0.000 deg,	R =    90.000 deg
};
P[9686]{
   GP1:
	UF : 1, UT : 1,		CONFIG : 'N U T, 0, 0, 1',
	X =  97.000  mm,	Y =  208.000  mm,	Z =   0.600 mm,
	W =180.000 deg,	P =   0.000 deg,	R =    90.000 deg
};
P[9687]{
   GP1:
	UF : 1, UT : 1,		CONFIG : 'N U T, 0, 0, 1',
	X =  97.000  mm,	Y =  208.000  mm,	Z =   15.000 mm,
	W =180.000 deg,	P =   0.000 deg,	R =    90.000 deg
};
P[9688]{
   GP1:
	UF : 1, UT : 1,		CONFIG : 'N U T, 0, 0, 1',
	X =  100.000  mm,	Y =  208.000  mm,	Z =   15.000 mm,
	W =180.000 deg,	P =   0.000 deg,	R =    90.000 deg
};
P[9689]{
   GP1:
	UF : 1, UT : 1,		CONFIG : 'N U T, 0, 0, 1',
	X =  100.000  mm,	Y =  208.000  mm,	Z =   0.600 mm,
	W =180.000 deg,	P =   0.000 deg,	R =    90.000 deg
};
P[9690]{
   GP1:
	UF : 1, UT : 1,		CONFIG : 'N U T, 0, 0, 1',
	X =  100.000  mm,	Y =  208.000  mm,	Z =   15.000 mm,
	W =180.000 deg,	P =   0.000 deg,	R =    90.000 deg
};
P[9691]{
   GP1:
	UF : 1, UT : 1,		CONFIG : 'N U T, 0, 0, 1',
	X =  103.000  mm,	Y =  208.000  mm,	Z =   15.000 mm,
	W =180.000 deg,	P =   0.000 deg,	R =    90.000 deg
};
P[9692]{
   GP1:
	UF : 1, UT : 1,		CONFIG : 'N U T, 0, 0, 1',
	X =  103.000  mm,	Y =  208.000  mm,	Z =   0.600 mm,
	W =180.000 deg,	P =   0.000 deg,	R =    90.000 deg
};
P[9693]{
   GP1:
	UF : 1, UT : 1,		CONFIG : 'N U T, 0, 0, 1',
	X =  103.000  mm,	Y =  208.000  mm,	Z =   15.000 mm,
	W =180.000 deg,	P =   0.000 deg,	R =    90.000 deg
};
P[9694]{
   GP1:
	UF : 1, UT : 1,		CONFIG : 'N U T, 0, 0, 1',
	X =  106.000  mm,	Y =  208.000  mm,	Z =   15.000 mm,
	W =180.000 deg,	P =   0.000 deg,	R =    90.000 deg
};
P[9695]{
   GP1:
	UF : 1, UT : 1,		CONFIG : 'N U T, 0, 0, 1',
	X =  106.000  mm,	Y =  208.000  mm,	Z =   0.600 mm,
	W =180.000 deg,	P =   0.000 deg,	R =    90.000 deg
};
P[9696]{
   GP1:
	UF : 1, UT : 1,		CONFIG : 'N U T, 0, 0, 1',
	X =  106.000  mm,	Y =  208.000  mm,	Z =   15.000 mm,
	W =180.000 deg,	P =   0.000 deg,	R =    90.000 deg
};
P[9697]{
   GP1:
	UF : 1, UT : 1,		CONFIG : 'N U T, 0, 0, 1',
	X =  109.000  mm,	Y =  208.000  mm,	Z =   15.000 mm,
	W =180.000 deg,	P =   0.000 deg,	R =    90.000 deg
};
P[9698]{
   GP1:
	UF : 1, UT : 1,		CONFIG : 'N U T, 0, 0, 1',
	X =  109.000  mm,	Y =  208.000  mm,	Z =   0.600 mm,
	W =180.000 deg,	P =   0.000 deg,	R =    90.000 deg
};
P[9699]{
   GP1:
	UF : 1, UT : 1,		CONFIG : 'N U T, 0, 0, 1',
	X =  109.000  mm,	Y =  208.000  mm,	Z =   15.000 mm,
	W =180.000 deg,	P =   0.000 deg,	R =    90.000 deg
};
P[9700]{
   GP1:
	UF : 1, UT : 1,		CONFIG : 'N U T, 0, 0, 1',
	X =  112.000  mm,	Y =  208.000  mm,	Z =   15.000 mm,
	W =180.000 deg,	P =   0.000 deg,	R =    90.000 deg
};
P[9701]{
   GP1:
	UF : 1, UT : 1,		CONFIG : 'N U T, 0, 0, 1',
	X =  112.000  mm,	Y =  208.000  mm,	Z =   0.600 mm,
	W =180.000 deg,	P =   0.000 deg,	R =    90.000 deg
};
P[9702]{
   GP1:
	UF : 1, UT : 1,		CONFIG : 'N U T, 0, 0, 1',
	X =  112.000  mm,	Y =  208.000  mm,	Z =   15.000 mm,
	W =180.000 deg,	P =   0.000 deg,	R =    90.000 deg
};
P[9703]{
   GP1:
	UF : 1, UT : 1,		CONFIG : 'N U T, 0, 0, 1',
	X =  115.000  mm,	Y =  208.000  mm,	Z =   15.000 mm,
	W =180.000 deg,	P =   0.000 deg,	R =    90.000 deg
};
P[9704]{
   GP1:
	UF : 1, UT : 1,		CONFIG : 'N U T, 0, 0, 1',
	X =  115.000  mm,	Y =  208.000  mm,	Z =   0.600 mm,
	W =180.000 deg,	P =   0.000 deg,	R =    90.000 deg
};
P[9705]{
   GP1:
	UF : 1, UT : 1,		CONFIG : 'N U T, 0, 0, 1',
	X =  115.000  mm,	Y =  208.000  mm,	Z =   15.000 mm,
	W =180.000 deg,	P =   0.000 deg,	R =    90.000 deg
};
P[9706]{
   GP1:
	UF : 1, UT : 1,		CONFIG : 'N U T, 0, 0, 1',
	X =  118.000  mm,	Y =  208.000  mm,	Z =   15.000 mm,
	W =180.000 deg,	P =   0.000 deg,	R =    90.000 deg
};
P[9707]{
   GP1:
	UF : 1, UT : 1,		CONFIG : 'N U T, 0, 0, 1',
	X =  118.000  mm,	Y =  208.000  mm,	Z =   0.600 mm,
	W =180.000 deg,	P =   0.000 deg,	R =    90.000 deg
};
P[9708]{
   GP1:
	UF : 1, UT : 1,		CONFIG : 'N U T, 0, 0, 1',
	X =  118.000  mm,	Y =  208.000  mm,	Z =   15.000 mm,
	W =180.000 deg,	P =   0.000 deg,	R =    90.000 deg
};
P[9709]{
   GP1:
	UF : 1, UT : 1,		CONFIG : 'N U T, 0, 0, 1',
	X =  121.000  mm,	Y =  208.000  mm,	Z =   15.000 mm,
	W =180.000 deg,	P =   0.000 deg,	R =    90.000 deg
};
P[9710]{
   GP1:
	UF : 1, UT : 1,		CONFIG : 'N U T, 0, 0, 1',
	X =  121.000  mm,	Y =  208.000  mm,	Z =   0.600 mm,
	W =180.000 deg,	P =   0.000 deg,	R =    90.000 deg
};
P[9711]{
   GP1:
	UF : 1, UT : 1,		CONFIG : 'N U T, 0, 0, 1',
	X =  121.000  mm,	Y =  208.000  mm,	Z =   15.000 mm,
	W =180.000 deg,	P =   0.000 deg,	R =    90.000 deg
};
P[9712]{
   GP1:
	UF : 1, UT : 1,		CONFIG : 'N U T, 0, 0, 1',
	X =  124.000  mm,	Y =  208.000  mm,	Z =   15.000 mm,
	W =180.000 deg,	P =   0.000 deg,	R =    90.000 deg
};
P[9713]{
   GP1:
	UF : 1, UT : 1,		CONFIG : 'N U T, 0, 0, 1',
	X =  124.000  mm,	Y =  208.000  mm,	Z =   0.600 mm,
	W =180.000 deg,	P =   0.000 deg,	R =    90.000 deg
};
P[9714]{
   GP1:
	UF : 1, UT : 1,		CONFIG : 'N U T, 0, 0, 1',
	X =  124.000  mm,	Y =  208.000  mm,	Z =   15.000 mm,
	W =180.000 deg,	P =   0.000 deg,	R =    90.000 deg
};
P[9715]{
   GP1:
	UF : 1, UT : 1,		CONFIG : 'N U T, 0, 0, 1',
	X =  127.000  mm,	Y =  208.000  mm,	Z =   15.000 mm,
	W =180.000 deg,	P =   0.000 deg,	R =    90.000 deg
};
P[9716]{
   GP1:
	UF : 1, UT : 1,		CONFIG : 'N U T, 0, 0, 1',
	X =  127.000  mm,	Y =  208.000  mm,	Z =   0.600 mm,
	W =180.000 deg,	P =   0.000 deg,	R =    90.000 deg
};
P[9717]{
   GP1:
	UF : 1, UT : 1,		CONFIG : 'N U T, 0, 0, 1',
	X =  127.000  mm,	Y =  208.000  mm,	Z =   15.000 mm,
	W =180.000 deg,	P =   0.000 deg,	R =    90.000 deg
};
P[9718]{
   GP1:
	UF : 1, UT : 1,		CONFIG : 'N U T, 0, 0, 1',
	X =  130.000  mm,	Y =  208.000  mm,	Z =   15.000 mm,
	W =180.000 deg,	P =   0.000 deg,	R =    90.000 deg
};
P[9719]{
   GP1:
	UF : 1, UT : 1,		CONFIG : 'N U T, 0, 0, 1',
	X =  130.000  mm,	Y =  208.000  mm,	Z =   0.600 mm,
	W =180.000 deg,	P =   0.000 deg,	R =    90.000 deg
};
P[9720]{
   GP1:
	UF : 1, UT : 1,		CONFIG : 'N U T, 0, 0, 1',
	X =  130.000  mm,	Y =  208.000  mm,	Z =   15.000 mm,
	W =180.000 deg,	P =   0.000 deg,	R =    90.000 deg
};
P[9721]{
   GP1:
	UF : 1, UT : 1,		CONFIG : 'N U T, 0, 0, 1',
	X =  133.000  mm,	Y =  208.000  mm,	Z =   15.000 mm,
	W =180.000 deg,	P =   0.000 deg,	R =    90.000 deg
};
P[9722]{
   GP1:
	UF : 1, UT : 1,		CONFIG : 'N U T, 0, 0, 1',
	X =  133.000  mm,	Y =  208.000  mm,	Z =   0.600 mm,
	W =180.000 deg,	P =   0.000 deg,	R =    90.000 deg
};
P[9723]{
   GP1:
	UF : 1, UT : 1,		CONFIG : 'N U T, 0, 0, 1',
	X =  133.000  mm,	Y =  208.000  mm,	Z =   15.000 mm,
	W =180.000 deg,	P =   0.000 deg,	R =    90.000 deg
};
P[9724]{
   GP1:
	UF : 1, UT : 1,		CONFIG : 'N U T, 0, 0, 1',
	X =  136.000  mm,	Y =  208.000  mm,	Z =   15.000 mm,
	W =180.000 deg,	P =   0.000 deg,	R =    90.000 deg
};
P[9725]{
   GP1:
	UF : 1, UT : 1,		CONFIG : 'N U T, 0, 0, 1',
	X =  136.000  mm,	Y =  208.000  mm,	Z =   0.600 mm,
	W =180.000 deg,	P =   0.000 deg,	R =    90.000 deg
};
P[9726]{
   GP1:
	UF : 1, UT : 1,		CONFIG : 'N U T, 0, 0, 1',
	X =  136.000  mm,	Y =  208.000  mm,	Z =   15.000 mm,
	W =180.000 deg,	P =   0.000 deg,	R =    90.000 deg
};
P[9727]{
   GP1:
	UF : 1, UT : 1,		CONFIG : 'N U T, 0, 0, 1',
	X =  139.000  mm,	Y =  208.000  mm,	Z =   15.000 mm,
	W =180.000 deg,	P =   0.000 deg,	R =    90.000 deg
};
P[9728]{
   GP1:
	UF : 1, UT : 1,		CONFIG : 'N U T, 0, 0, 1',
	X =  139.000  mm,	Y =  208.000  mm,	Z =   0.600 mm,
	W =180.000 deg,	P =   0.000 deg,	R =    90.000 deg
};
P[9729]{
   GP1:
	UF : 1, UT : 1,		CONFIG : 'N U T, 0, 0, 1',
	X =  139.000  mm,	Y =  208.000  mm,	Z =   15.000 mm,
	W =180.000 deg,	P =   0.000 deg,	R =    90.000 deg
};
P[9730]{
   GP1:
	UF : 1, UT : 1,		CONFIG : 'N U T, 0, 0, 1',
	X =  142.000  mm,	Y =  208.000  mm,	Z =   15.000 mm,
	W =180.000 deg,	P =   0.000 deg,	R =    90.000 deg
};
P[9731]{
   GP1:
	UF : 1, UT : 1,		CONFIG : 'N U T, 0, 0, 1',
	X =  142.000  mm,	Y =  208.000  mm,	Z =   0.600 mm,
	W =180.000 deg,	P =   0.000 deg,	R =    90.000 deg
};
P[9732]{
   GP1:
	UF : 1, UT : 1,		CONFIG : 'N U T, 0, 0, 1',
	X =  142.000  mm,	Y =  208.000  mm,	Z =   15.000 mm,
	W =180.000 deg,	P =   0.000 deg,	R =    90.000 deg
};
P[9733]{
   GP1:
	UF : 1, UT : 1,		CONFIG : 'N U T, 0, 0, 1',
	X =  145.000  mm,	Y =  208.000  mm,	Z =   15.000 mm,
	W =180.000 deg,	P =   0.000 deg,	R =    90.000 deg
};
P[9734]{
   GP1:
	UF : 1, UT : 1,		CONFIG : 'N U T, 0, 0, 1',
	X =  145.000  mm,	Y =  208.000  mm,	Z =   0.600 mm,
	W =180.000 deg,	P =   0.000 deg,	R =    90.000 deg
};
P[9735]{
   GP1:
	UF : 1, UT : 1,		CONFIG : 'N U T, 0, 0, 1',
	X =  145.000  mm,	Y =  208.000  mm,	Z =   15.000 mm,
	W =180.000 deg,	P =   0.000 deg,	R =    90.000 deg
};
P[9736]{
   GP1:
	UF : 1, UT : 1,		CONFIG : 'N U T, 0, 0, 1',
	X =  148.000  mm,	Y =  208.000  mm,	Z =   15.000 mm,
	W =180.000 deg,	P =   0.000 deg,	R =    90.000 deg
};
P[9737]{
   GP1:
	UF : 1, UT : 1,		CONFIG : 'N U T, 0, 0, 1',
	X =  148.000  mm,	Y =  208.000  mm,	Z =   0.600 mm,
	W =180.000 deg,	P =   0.000 deg,	R =    90.000 deg
};
P[9738]{
   GP1:
